(* LS Electric XG5000 project: QT(230517) *)
(* PLC NewPLC *)
(* module base 0 slot 0: FEnet:XGL-EFMT(B) (Fast Ethernet 통신 모듈, 전기 Master) *)
(* module base 1 slot 0: 아날로그입력 모듈:XGF-AC8A (A/D 전류 입력형 8채널) *)
(* module base 1 slot 1: 입력 모듈:XGI-D28A/B (DC 24V 입력, 64점 (전류소스 싱크공용/ 전류소스 입력)) *)
(* module base 1 slot 2: 입력 모듈:XGI-D28A/B (DC 24V 입력, 64점 (전류소스 싱크공용/ 전류소스 입력)) *)
(* module base 1 slot 3: 출력 모듈:XGQ-TR8A/B (트랜지스터 출력, 64점 (0.1A용, 싱크출력/소스출력)) *)
(* module base 1 slot 4: 출력 모듈:XGQ-TR8A/B (트랜지스터 출력, 64점 (0.1A용, 싱크출력/소스출력)) *)
(* module base 1 slot 5: Cnet:XGL-CH2A/B (Cnet 통신 모듈(RS-232C, RS-422/485)) *)
VAR_GLOBAL
    C485 : TON;
    C486 : TON;
    C487 : TON;
    TCPIP : TON;
    _0000_STAND_ALONE AT %LX60144 : BOOL; (* FEnet: 연결 안된 상태(Ver 6.0이상) *)
    _0100_CH0_ACT AT %UX1.0.16 : BOOL; (* 아날로그입력 모듈: 채널0 운전중 *)
    _0100_CH0_DATA AT %UW1.0.2 : INT; (* 아날로그입력 모듈: 채널0 변환값 *)
    _0100_CH0_IDD AT %UX1.0.160 : BOOL; (* 아날로그입력 모듈: 채널0 입력단선검출 *)
    _0100_CH1_ACT AT %UX1.0.17 : BOOL; (* 아날로그입력 모듈: 채널1 운전중 *)
    _0100_CH1_DATA AT %UW1.0.3 : INT; (* 아날로그입력 모듈: 채널1 변환값 *)
    _0100_CH1_IDD AT %UX1.0.161 : BOOL; (* 아날로그입력 모듈: 채널1 입력단선검출 *)
    _0100_CH2_ACT AT %UX1.0.18 : BOOL; (* 아날로그입력 모듈: 채널2 운전중 *)
    _0100_CH2_DATA AT %UW1.0.4 : INT; (* 아날로그입력 모듈: 채널2 변환값 *)
    _0100_CH2_IDD AT %UX1.0.162 : BOOL; (* 아날로그입력 모듈: 채널2 입력단선검출 *)
    _0100_CH3_ACT AT %UX1.0.19 : BOOL; (* 아날로그입력 모듈: 채널3 운전중 *)
    _0100_CH3_DATA AT %UW1.0.5 : INT; (* 아날로그입력 모듈: 채널3 변환값 *)
    _0100_CH3_IDD AT %UX1.0.163 : BOOL; (* 아날로그입력 모듈: 채널3 입력단선검출 *)
    _0100_CH4_ACT AT %UX1.0.20 : BOOL; (* 아날로그입력 모듈: 채널4 운전중 *)
    _0100_CH4_DATA AT %UW1.0.6 : INT; (* 아날로그입력 모듈: 채널4 변환값 *)
    _0100_CH4_IDD AT %UX1.0.164 : BOOL; (* 아날로그입력 모듈: 채널4 입력단선검출 *)
    _0100_CH5_ACT AT %UX1.0.21 : BOOL; (* 아날로그입력 모듈: 채널5 운전중 *)
    _0100_CH5_DATA AT %UW1.0.7 : INT; (* 아날로그입력 모듈: 채널5 변환값 *)
    _0100_CH5_IDD AT %UX1.0.165 : BOOL; (* 아날로그입력 모듈: 채널5 입력단선검출 *)
    _0100_CH6_ACT AT %UX1.0.22 : BOOL; (* 아날로그입력 모듈: 채널6 운전중 *)
    _0100_CH6_DATA AT %UW1.0.8 : INT; (* 아날로그입력 모듈: 채널6 변환값 *)
    _0100_CH6_IDD AT %UX1.0.166 : BOOL; (* 아날로그입력 모듈: 채널6 입력단선검출 *)
END_VAR

(* Comments on direct variables
%IX1.1.0	TK-301 HLV-PB
%IX1.1.1	P301ATR
%IX1.1.2	P301A Local sw
%IX1.1.3	P12AB
%IX1.1.4	LPB1AO
%IX1.1.5	P301A stop-PB
%IX1.1.6	P301A run-PB
%IX1.1.7	P301BTR
%IX1.1.8	P301B Local sw
%IX1.1.9	LPB1BF
%IX1.1.10	LPB1BO
%IX1.1.11	P301B stop-PB
%IX1.1.12	P301B Run PB
%IX1.1.13	P301CTR
%IX1.1.14	P301C Local sw
%IX1.1.15	LPB1CF
%IX1.1.16	LPB1CO
%IX1.1.17	P301C stop-PB
%IX1.1.18	P301C Run PB
%IX1.1.19	TK301-Clearance
%IX1.1.20	TK301-LEK
%IX1.1.21	P301ATH
%IX1.1.22	P301BTH
%IX1.1.23	P301CTH
%IX1.1.24	PUMP Room
%IX1.1.25	TK-302 HLV-PB
%IX1.1.26	  P302A  Trouble
%IX1.1.27	 P302A  LOCAL SW
%IX1.1.28	LPB2AF
%IX1.1.29	LPB2AO
%IX1.1.30	P302A stop-PB
%IX1.1.31	P302A run-PB
%IX1.1.32	  P302B  Trouble
%IX1.1.33	 P302B  LOCAL SW
%IX1.1.34	LPB2BF
%IX1.1.35	LPB2BO
%IX1.1.36	P302B stop-PB
%IX1.1.37	P302B run-PB
%IX1.1.38	  P302C  Trouble
%IX1.1.39	P302C  Local SW
%IX1.1.40	LPB2CF
%IX1.1.41	LPB2CO
%IX1.1.42	P302C stop-PB
%IX1.1.43	P302C run-PB
%IX1.1.44	TK302-Clearance
%IX1.1.45	TK302-LEK
%IX1.1.46	P302ATH
%IX1.1.47	P302BTH
%IX1.1.48	P302CTH
%IX1.1.49	TK-302 EM
%IX1.1.50	HLVD
(H30201)
%IX1.1.51	W30201
%IX1.1.52	  P303  Trouble
%IX1.1.53	P303  Local SW
%IX1.1.54	EMS1X
%IX1.1.55	EMS2X
%IX1.1.56	P303 stop-PB
%IX1.1.57	P303 Run PB
%IX1.1.58	Drain-303
Clearance
%IX1.1.59	EMS3X
%IX1.1.60	EMS4X
%IX1.1.61	P301A  1차 선택 SWITCH  (PANEL)
%IX1.1.62	P301B 1차 선택 SWITCH  (PANEL)
%IX1.1.63	P302A 1차 선택 SWITCH  (PANEL)
%IX1.2.0	P302B 1차 선택 SWITCH  (PANEL)
%IX1.2.1	P-301A 2차-PB
%IX1.2.2	P-301B 2차-PB
%IX1.2.3	P-302A 2차-PB
%IX1.2.4	P-302B 2차-PB
%IX1.2.5	Power-off PB
%IX1.2.6	Power-on PB
%IX1.2.7	Manual-PB
%IX1.2.8	Auto-PB
%IX1.2.9	AUTO START P/B
%IX1.2.10	Lamp-test PB
%IX1.2.11	AUTO STOP (PANEL)
%IX1.2.12	Horn Stop Panel
%IX1.2.13	EM_Reset
[Panel]
%IX1.2.14	PLC-Stanby operation
%IX1.2.16	운전선택 SCADA OR PANEL
%IX1.2.17	PANEL EM
%IX1.2.18	EMS1_C22
%IX1.2.19	EMS2_C21
%IX1.2.20	EMS3_C20
%IX1.2.21	EMS4_C19
%IX1.2.22	Cam1_R1
%IX1.2.23	Cam2_R2
%IX1.2.24	Cam3_R3
%IX1.2.25	BCVF
%IX1.2.26	TLV1
%IX1.2.27	TLV2
%IX1.2.28	TLV3
%IX1.2.29	TLV4
%IX1.2.32	SHELTURN1 TLV
%IX1.2.33	SHELTURN2 TLV
%IX1.2.34	SHELTURN3 TLV
%IX1.2.35	SHELTURN4 TLV
%IX1.2.36	P301A FS 
%IX1.2.37	P301B FS 
%IX1.2.38	P301C FS 
%IX1.2.39	P302A FS 
%IX1.2.40	P302B FS 
%IX1.2.41	P302C FS 
%IX1.2.42	P303 FS 
%IX1.2.43	P301A MC ON SIG 
%IX1.2.44	P301B MC ON SIG 
%IX1.2.45	P301C MC ON SIG 
%IX1.2.46	P302A MC ON SIG 
%IX1.2.47	P302B MC ON SIG 
%IX1.2.48	P302C MC ON SIG 
%IX1.2.49	P303 MC ON SIG 
%IX1.2.56	HLVB(하차 VALVE)
%IX1.3.0	PL29-R
%IX1.3.1	L37-Y
%IX1.3.48	TK-110 HLV 선택PB
%IX2.3.1	P101A THERMOSTAT
%ID1.0.0	디지털_입력
%QX1.3.0	TK-301 HLV on
%QX1.3.1	P301A Trouble
%QX1.3.2	  P301A  Local
%QX1.3.3	P301A-stop Lamp
%QX1.3.4	P301A Run
%QX1.3.5	P301B-Trouble
%QX1.3.6	P301B- Local
%QX1.3.7	P301B-stop
%QX1.3.8	P301B Run
%QX1.3.9	P301C-Trouble
%QX1.3.10	P301C- Local
%QX1.3.11	P301C-stop Lamp
%QX1.3.12	P301C Run
%QX1.3.13	TK-301 HH
%QX1.3.14	TK-301 H
%QX1.3.15	TK-301 ATG TROUBLE
%QX1.3.16	TK-301 L
%QX1.3.17	TK-301 LL
%QX1.3.18	TK-301 Leakage
%QX1.3.19	TK-302 HLV on
%QX1.3.20	P302A Trouble
%QX1.3.21	  P302A   Local
%QX1.3.22	P302A  Stop Lamp
%QX1.3.23	P302A Run
%QX1.3.24	P302B-Trouble
%QX1.3.25	  P302B   Local
%QX1.3.26	P302B  Stop Lamp
%QX1.3.27	P302B Run
%QX1.3.28	P302C-Trouble
%QX1.3.29	  P302C  Local
%QX1.3.30	P302C  Stop Lamp
%QX1.3.31	P302C Run
%QX1.3.32	TK-302 HH
%QX1.3.33	TK-302 H
%QX1.3.34	TK-302 ATG TROUBLE
%QX1.3.35	TK-302 L
%QX1.3.36	TK-302 LL
%QX1.3.37	TK-302 Leakage
%QX1.3.38	TK-303 HLVD
%QX1.3.39	TK-303 Water
%QX1.3.40	P303-Trouble lamp
%QX1.3.41	  P303  Local
%QX1.3.42	P303  Stop Lamp
%QX1.3.43	P303 Run
%QX1.3.44	TK-303 Max2
%QX1.3.45	TK-303_LT33_H
%QX1.3.46	TK-303 Nomal
%QX1.3.47	TK-303 Min1
%QX1.3.48	TK-303 Min2
%QX1.3.49	P301A 1차 선택 Lamp
%QX1.3.50	P301A 2차 선택 Lamp
%QX1.3.51	P301B 1차 선택 Lamp
%QX1.3.52	P301B 2차 선택 Lamp
%QX1.3.53	P302A 1차 선택 Lamp
%QX1.3.54	P302A 2차 선택 Lamp
%QX1.3.55	P302B 1차 선택 Lamp
%QX1.3.56	P302B 2차 선택 Lamp
%QX1.3.57	Power-off LAMP
%QX1.3.58	Power-on LAMP
%QX1.3.59	Manual LAMP
%QX1.3.60	Auto 선택 LAMP
%QX1.3.61	AUTO START LAMP
%QX1.3.62	AUTO STOP LAMP
%QX1.3.63	압력저하 (PT-301)
%QX1.4.0	Horn Stop Lamp
%QX1.4.1	Pump-start 6time/h
%QX1.4.2	BPCV1-Lamp
%QX1.4.3	CVP-Lamp
%QX1.4.4	EV-Lamp
%QX1.4.5	EM RESET LAMP
%QX1.4.6	BCVF-Lamp
%QX1.4.7	Lamp_test LAMP
%QX1.4.8	PUMP Room
%QX1.4.9	EM-Panel
%QX1.4.10	Shelter-1
%QX1.4.11	Shelter-2
%QX1.4.12	Shelter-3
%QX1.4.13	Shelter-4
%QX1.4.14	Emergency-local
%QX1.4.15	PIT1-Trouble 
%QX1.4.16	PIT2-Trouble 
%QX1.4.17	FIT1-Trouble 
%QX1.4.18	FIT2-Trouble 
%QX1.4.19	FIT3-Trouble 
%QX1.4.20	FIT4-Trouble 
%QX1.4.21	MASTER PLC LAMP
%QX1.4.22	Control-unit 1 Trouble
%QX1.4.23	STANDBY PLC LAMP
%QX1.4.24	Control-unit 2 Trouble
%QX1.4.25	Horn Relay
%QX1.4.26	PUMP Room
%QX1.4.27	TK-302 EM
%QX1.4.28	Panel 선택 Lamp
%QX1.4.29	SCADA 선택 Lamp
%QX1.4.30	BPCV1-Sol
%QX1.4.31	BPCV2-Sol
%QX1.4.32	CVP SOL
%QX1.4.33	EV-Sol
%QX1.4.34	R1_PT3-4/PT5-6
%QX1.4.35	R2_FT1-2/FT5-6
%QX1.4.36	R2_FT3-4/FTT-8
%QX1.4.37	TK-301 HLV OPEN LAMP
%QX1.4.38	P301A Run LAMP
%QX1.4.39	P301B Run LAMP
%QX1.4.40	P301C Run LAMP
%QX1.4.41	TK-302 HLV OPEN LAMP
%QX1.4.42	P302A Run LAMP
%QX1.4.43	P302B Run LAMP
%QX1.4.44	P302C Run LAMP
%QX1.4.45	P303 Run LAMP
%QX1.6.2	SCADA 선택 Lamp
%QX1.6.3	Panel 선택 Lamp
%QX2.2.26	출하 PUMP P101A 1차 운전 선택 Lamp
%QX2.2.27	출하 PUMP P101B 1차 운전 선택 Lamp
%QX2.2.42	출하 PUMP P101A 2차 운전 선택 Lamp
%QX2.2.43	출하 PUMP P101B 2차 운전 선택 Lamp
%MX0	P301A_Run
%MX1	P301B_Run
%MX2	P301A_Pump
%MX3	P301A_FS
%MX5	P301A_Trouble
%MX6	TK-301 HLV,P301A,P301B_Run
%MX7	P301A,OR P301B_RUN
%MX8	P301B_Pump
%MX9	P301B_FS
%MX10	P301A_P301B_ Trouble
%MX12	BPCV_On
%MX14	P301B_Trouble
%MX15	P301C_RUN
%MX16	P301C_STOP
%MX17	P301C_PUMP
%MX18	QT_BOTTOM TAP COLOR(X PUMP RUN)
%MX19	TK-302 HLV,P302A,P302B_Run
%MX20	P302A_Run
%MX21	P302A,OR P302B_RUN
%MX22	P302A_Pump
%MX23	P302A_FS
%MX24	P302A_Trouble
%MX25	P302B_Run
%MX26	P302A_P302B_ Trouble
%MX27	P302B-Pump
%MX28	P302B_FS
%MX29	P302B_Trouble
%MX30	P302C_Run
%MX31	P301 회수중
%MX32	P302C_Pump
%MX33	P302C_FS
%MX34	P302C_Trouble
%MX35	P303_Run
%MX36	P302 회수중
%MX37	P303_Pump
%MX38	P303_FS
%MX39	P303_Trouble
%MX40	Alarm Reset
%MX45	TLV1
%MX46	TLV2
%MX47	TLV3
%MX48	TLV4
%MX49	HLV1
%MX50	HLV2
%MX51	TK-301 출하
%MX52	출하_EV
%MX53	출하_CVP
%MX54	출하_BPCV
%MX55	회수라인
%MX56	TK301_회수
%MX57	TK302_회수
%MX58	QT01_출하
%MX59	QT02_출하
%MX60	QT03_출하
%MX61	QT04_출하
%MX62	AUTO START OK
%MX65	TLV1
%MX66	TLV2
%MX67	TLV3
%MX68	TLV4
%MX79	TK-104 선택 SCADA    (수령)
%MX82	QT_TANK_HH
%MX100	TK-301 CH0 단선
%MX101	TK-301 Min2
%MX102	TK-301 Min1
%MX103	TK-301 Max1
%MX104	TK-301 Max2
%MX105	TK-302 CH1 단선
%MX106	TK-302 Min2
%MX107	TK-302 Min1
%MX108	TK-302 Max1
%MX109	TK-302 Max2
%MX110	TK-303 CH1 단선
%MX111	TK-303 Min2
%MX112	TK-303 Min1
%MX113	TK-303 Max1
%MX114	TK-303 Max2
%MX128	P301A run-PB  (SCADA)
%MX129	P301A stop-PB  (SCADA)
%MX130	Manual_Scada
%MX131	Auto_Scada
%MX132	P301B Run PB(SCADA)
%MX133	P301B stop-PB(SCADA)
%MX134	  AUTO   START  (SCADA)
%MX135	AUTO STOP (SCADA)
%MX136	P301C Run PB(SCADA)
%MX137	P301C stop-PB(SCADA)
%MX138	P302A Run PB(SCADA)
%MX139	P302A stop-PB(SCADA)
%MX140	P302B Run PB(SCADA)
%MX141	P302B stop-PB(SCADA)
%MX142	P302C Run PB(SCADA)
%MX143	P302C stop-PB(SCADA)
%MX144	P303 Run PB(SCADA)
%MX145	P303 stop-PB(SCADA)
%MX146	EM-Reset
[SCADA]
%MX147	Horn Stop SCADA
%MX148	P301A Lock key Run
%MX149	P301B Lock key Run
%MX150	P301C Lock key Run
%MX151	P302A Lock key Run
%MX152	P302B Lock key Run
%MX153	P302C Lock key Run
%MX154	P303 Lock key Run
%MX160	이글루#1유량 - 값
%MX161	이글루#2유량 - 값
%MX162	이글루#3유량 - 값
%MX163	이글루#4유량 - 값
%MX164	수령 유량 -값
%MX169	L5 BPCV
%MX170	L6 CVP
%MX171	L7 BCVF (By-Pass Valve)
%MX172	L8 EV
%MX173	수령유량 - 값
%MX177	TK-303_LT33_FAULT
%MX180	P303_Remote
%MX181	P303_Stop
%MX182	P303_Run
%MX183	P303_Fault
%MX184	P303_F.S
%MX185	P303_O.L
%MX186	P303_HLVD
%MX192	TK-301 HLV SCADA ON
%MX193	TK-302 HLV SCADA ON
%MX206	TK-301 ATG NO SIGNAL
%MX207	TK-301_LL
%MX208	TK-301_LT31_L
%MX209	TK-301_LT31_H
%MX210	TK-301_HH_SIG
%MX212	P301A_Key
%MX213	P301A_Remote
%MX214	P301A_Stop
%MX215	P301A_Run
%MX216	P301A_Fault
%MX217	P301A FS_Fault
%MX218	P301A_O.L
%MX219	P301B_Key
%MX220	301B_Remote
%MX221	P301B_Stop
%MX222	P301B_Run
%MX223	P301B_Fault
%MX224	P301B_F.S
%MX225	P301B_O.L
%MX226	P301C_Remote
%MX227	P301C_Stop
%MX228	P301C_Run
%MX229	P301C_Fault
%MX235	TK-302_LL
SIG
%MX236	TK-302 L
SIG
%MX237	TK-302_H
_SIG
%MX238	TK-302_HH_SIG
%MX239	TK-302 ATG NO SIGNAL
%MX240	P302A_Key
%MX241	P302A_Remote
%MX242	P302A_Stop
%MX243	P302A_Run
%MX244	P302A_Fault
%MX245	P302A_F.S
%MX246	P302A_O.L
%MX247	P302B_Key
%MX248	P302B_Remote
%MX249	P302B_Stop
%MX250	P302B_Run
%MX251	P302B_Fault
%MX252	P302B_F.S
%MX253	P302B_O.L
%MX254	P302C_Remote
%MX255	P302C_Stop
%MX256	P302C_Run
%MX257	P302C_Fault
%MX263	PRI1_301A
%MX264	PRI1_301B
%MX265	PRI1_302A
%MX266	PRI1_302B
%MX267	PRI2_301A
%MX268	PRI2_301B
%MX269	PRI2_302A
%MX270	PRI2_302B
%MX272	CH1 PIT3-4 Trouble
%MX273	CH2 FT301 Trouble
%MX274	CH3 FIT3-4 Trouble
%MX277	CH3 FT-302 Trouble
%MX301	P-301A 1차-out
%MX303	P-301B 1차-out
%MX305	P-302A 1차-out
%MX307	P-302B 1차-out
%MX309	P-301A 2차-out
%MX310	P-301B 2차-on
%MX312	P-302A 2차-on
%MX313	TANK101 LEVEL 15%   L
%MX314	P-302B 2차-on
%MX330	TK-303_HH
%MX331	TK-303_H
%MX332	TK-303_ATG TROUBLE
%MX333	TK-303_L
%MX334	TK-303_LL
%MX335	QT_NMR#3
SIGNAL OFF 
ALARM
%MX340	P301A 1차 선택
%MX341	P301B 1차 선택
%MX342	P302A 1차 선택
%MX343	P302B 1차 선택
%MX344	P301A 2차 선택
%MX345	P301B 2차 선택
%MX346	P302A 2차 선택
%MX347	P302B 2차 선택
%MX352	P012A 2차 선택
%MX353	P012B 2차 선택
%MX360	P012A 1차 선택
%MX361	P021B 1차 선택
%MX362	P021A 2차 선택
%MX363	P021B 2차 선택
%MX398	1차 펌프 작동
%MX399	1차 펌프정지 압력
%MX400	Auto Run SIG
%MX401	1차 펌프 정지
%MX402	1차 펌프 초기 기동 압력
%MX403	1차 회수유량
%MX404	2차 펌프 작동
%MX405	1차 회수유량
%MX406	2차 회수유량
%MX407	2차 펌프정지
%MX408	1차 정지유량
%MX409	1차 재기동방지
%MX412	2차 펌프 정지
%MX413	1차 펌프정지 SIG
%MX414	1차 펌프 정지
%MX448	P301A  1차 선택 SWITCH  (SCADA)
%MX449	P301B 1차 선택 SWITCH  (SCADA)
%MX450	P301A 2차 선택 SWITCH  (SCADA)
%MX451	P301B 2차 선택 SWITCH  (SCADA)
%MX452	P302A 1차 선택 SWITCH  (SCADA)
%MX453	P302B 1차 선택 SWITCH  (SCADA)
%MX454	P302A 2차 선택 SWITCH  (SCADA)
%MX455	P302B 2차 선택 SWITCH  (SCADA)
%MX456	선택완료  (SCADA)
%MX458	P012A  1차 선택 SWITCH  (SCADA)
%MX459	P012B  1차 선택 SWITCH  (SCADA)
%MX460	P012A  2차 선택 SWITCH  (SCADA)
%MX461	P012B  2차 선택 SWITCH  (SCADA)
%MX468	P021A  1차 선택 SWITCH  (SCADA)
%MX469	P021B 1차 선택 SWITCH  (SCADA)
%MX470	P021A  2차 선택 SWITCH  (SCADA)
%MX471	P021B 2차 선택 SWITCH  (SCADA)
%MX500	통신 쓰기 PULS
%MX501	통신 읽기 PULS
%MX511	Auto_ P-301A_ON_REQ
%MX512	Scada_auto
%MX513	Scada_man
%MX514	S-P301A manual Run
%MX515	S-P301B manual Run
%MX516	S-P301C manual Run
%MX517	S-P302A manual Run
%MX518	S-P302B manual Run
%MX519	S-P302C manual Run
%MX520	S-P303 manual Run
%MX528	Shelturn4-Em
%MX529	Total Emergency
%MX530	 Total Alarm
%MX531	Horn Stop
%MX532	TK-301 HLV on-off
%MX533	TK-302 HLV on-off
%MX534	CVP_on
%MX536	HLV21201 TK110 OPEN PULS(MANU)
%MX537	Any HLV Open
%MX538	TK-302 Interlock 
%MX539	TK-301 Interlock 
%MX543	P-301A 1차_off
%MX544	P-301A 1차_out
%MX545	P-301B 1차_off
%MX546	P-301B 1차_out
%MX547	P-302A 1차_off
%MX548	P-302A 1차_out
%MX549	P-302B 1차_off
%MX550	P-302B 1차_out
%MX551	P-301A 2차_off
%MX552	P-301A 2차_out
%MX553	P-301B 2차_off
%MX554	P-301B 2차_out
%MX555	P-302A 2차_off
%MX556	P-302A 2차_out
%MX557	P-302B 2차_off
%MX558	P-302B 2차_out
%MX561	TK301 Auto
1차 
펌프운전중 
%MX562	Auto-1차 펌프정지 
%MX563	TK301 Auto
2차 
펌프운전중 
%MX564	Auto-2차 펌프정지 
%MX565	Auto P-301A_ON
%MX566	Auto P-301B_ON
%MX567	Auto P-302A_ON
%MX568	Auto P-302B_ON
%MX581	TK302 Auto
1차 
펌프운전중 
%MX591	TK302 Auto
2차 
펌프운전중 
%MX592	Auto_2차 펌프정지
%MX593	자동운전 시작
%MX594	펌프정지 압력
%MX595	Auto Run
%MX596	자동운전 정지
%MX597	1-2차 펌프on
%MX598	2차 펌프준비
%MX599	2차 펌프on
%MX600	1차 회수유량
%MX601	2차 회수유량
%MX602	2차 펌프정지
%MX603	1차 정지유량
%MX604	1차 재기동방지
%MX605	2차 펌프정지
%MX606	1차 펌프정지
%MX607	펌프운전 Rest
%MX640	PUMP Room
%MX641	TK-302 Em 사용안함
%MX642	TK-301 & 302 Em
%MX643	Panel-Em
%MX644	Shelturn1-Em
%MX645	Shelturn2-Em
%MX646	Shelturn3-Em
%MX647	Shelturn4-C19
%MX648	Local EM
%MX649	EMS1X
%MX650	EMS2X
%MX651	EMS3X
%MX652	EMS4X
%MX656	RS-485 통신이상
%MX657	TCPIP 통신이상
%MX1010	모드버스 브럭1-1 동작
%MX1200	모드버스 브럭2-1 동작
%MX1220	모드버스 브럭2-2 동작
%MX1300	모드버스 브럭3-1 동작
%MX1320	모드버스 브럭3-2 동작
%MX1400	모드버스 브럭4-1 동작
%MX1420	모드버스 브럭4-2 동작
%MX1500	모드버스 브럭5-1 동작
%MX1520	모드버스 브럭5-2 동작
%MX3232	이중화운전_A_Side_MASTER
%MX3233	이중화운전_B_Side_MASTER
%MX3234	A-Side 단독운전
%MX3235	B-Side 단독운전
%MX4816	AUTO HLV_301 OPEN
%MX4832	AUTO HLV_302 OPEN
%MX6400	Panel Manual
%MX6401	SCADA Manual
%MX6402	Panel Auto
%MX6403	SCADA Auto
%MX6405	BUZZER STOP
%MX6410	Manual 선택
%MX6411	Auto 선택
%MX6464	LAMP TEST SIG
%MX6476	MAIN PNL-EM
%MX10002	TEST2
%MX12800	AUTO START OK
%MX12801	AUTO STOP OK
%MX19200	P301A ALARM
%MX19201	P301A FS ALARM
%MX19202	P301B ALARM
%MX19203	P301B FS ALARM
%MX19204	P301C ALARM
%MX19205	P301C FS ALARM
%MX19206	P302A ALARM
%MX19207	P302A FS ALARM
%MX19208	P302B ALARM
%MX19209	P302B FS ALARM
%MX19210	P302C ALARM
%MX19211	P302C FS ALARM
%MX19212	P303 
ALARM
%MX19213	P303 FS ALARM
%MX19215	P301A FS SIG
%MX19216	P301B FS SIG
%MX19217	P301C FS SIG
%MX19218	P302A FS SIG
%MX19219	P302B FS SIG
%MX19220	P302C FS SIG
%MX19221	P303 FS SIG
%MX19264	P301A 수동 RUN
%MX19265	P301B 수동 RUN
%MX19266	P301C 수동 RUN
%MX19267	P302A 수동 RUN
%MX19268	P302B 수동 RUN
%MX19269	P302C 수동 RUN
%MX19270	P303 수동 RUN
%MX19905	P301A 1차 작동
%MX19906	P301A 2차 작동
%MX19969	P301B 1차 작동
%MX19970	P301B 2차 작동
%MX20545	P302A 1차 작동
%MX20546	P302A 2차 작동
%MX20609	P302B 1차 작동
%MX20610	P302B 2차 작동
%MX23087	Auto start all ready
%MX23089	ARES Stop SIG
%MX23680	TK-301 수령 송유관 색변화
%MX23681	TK-301  불출 송유관 색변화
%MX23682	TK-301,302 수령 송유관 색변화 
%MX23683	TK-301,302 불출 송유관 색변화
%MX23684	TK-302 수령 송유관 색변화
%MX23685	TK-302 불출 송유관 색변화 2
%MX23686	TK-301C,302C DRAIN 송유관 색변화
%MX23687	TK-302 DRAIN 송유관 색변화
%MX23688	SHELTURN1 송유관 색변화1 
%MX23689	SHELTURN2 송유관 색변화 2
%MX23690	SHELTURN3 송유관 색변화
%MX23691	SHELTURN4 송유관 색변화
%MX25600	AUTO START OK
%MX25602	ALL REMOTE
%MX25665	P101A Auto 2차 Run
%MX25666	P101B Auto 1차 Run
%MX25667	P101B Auto 2차 Run
%MX26112	QT_Auto_2st_Pump Run
%MX26113	QT_Auto_restart_alarm[TLV_SIG]
%MX26240	1차 PUMP Running Timing
%MX26241	2차 PUMP Running Timing
%MX26242	1차 PUMP Stoping
%MX26243	2차 PUMP Stoping
%MX26244	Auto Run BPCV Stop
%MX26246	1차 펌프 정지조건 홀딩
%MX26247	헌팅 보정
%MX26250	1차 PUMP Stoping 조건
%MX26256	holding pressure charge
%WW0	C22_BCU STATUS
%WW1	C22 BCU STATUS VALUE
%WW2	C21_BCU STATUS
%WW3	C20 BCU STATUS VALUE
%WW4	C20 BCU STATUS
%WW5	C20 BCU STATUS VALUE
%WW6	C19 BCU STATUS
%WW7	C19 BCU STATUS VALUE
%WW10	 P301 1차 선택 SET
%WW11	1차 선택 SET
%WW12	2차 선택 SET
%WW13	 P302 2차 선택 SET
%WW20	TANK301 문자열
%WW21	TK-302 문자열
%WW102	TK-301 LEVEL (PLC -> SCADA)
%WW150	P301A RUN SET
%WW151	P301B RUN SET
%WW152	P301C RUN SET
%WW153	P302A RUN SET
%WW154	P302B RUN SET
%WW155	P302C RUN SET
%WW156	P303 RUN SET
%WW202	TK-302 LEVEL (PLC -> SCADA)
%WW211	TK-112 H SET
%WW310	TK-301 HH SET
%WW311	TK-301 H SET
%WW312	TK-301 L SET
%WW313	TK-301 LL SET
%WW320	TK-302 HH SET
%WW321	TK-302 H SET
%WW322	TK-302 L SET
%WW323	TK-302 LL SET
%WW330	TK-303 HH SET
%WW331	TK-303 H SET
%WW332	TK-303 L SET
%WW333	TK-303 LL SET
%WW440	불출유량 - 회수유량 = 값
%WW500	TK301Level NRM500 - >PLC
%WW501	Error Status Ref.TK301
[NMR#3]
word
%WW503	TK302Level(NRM5000 ->PLC)
%WW504	Error Status Ref.TK302
[NMR#3]
word
%WW506	DRAIN TANK TK-111 LEVEL (PLC -> SCADA)
%WW682	TK-301 VOLUME (CTM->PLC)
%WW690	TK303 VOLUME(커텀스->PLC)
%WW691	TK111 VOLUME(커텀스->PLC)
%WW1000	이글루 #1 유량(High)
%WW1001	이글루 #1 유량(Low)
%WW1020	이글루 #2 유량(High)
%WW1021	이글루 #2 유량(Low)
%WW1040	이글루 #3 유량(High)
%WW1041	이글루 #3 유량 (Low)
%WW1060	이글루 #4 유량(high)
%WW1061	이글루 #4 유량(Low)
%WW1080	수령 유량
(High)
%WW1081	수령 유량 (Low)
%WW1100	PT301 출하압력 값
%WW1102	PT301출하압력 PSI
%WW1200	FT301 출하유량 값
%WW1202	FT301출하유량 GPM
%WW1204	FT301 출하유량
%WW1300	FT302 회수유량 값
%WW1302	FT302회수유량 GPM
%WW1304	FT302 회수유량
%WW1400	TK_303 변환값
%WW1402	TK-303 LEVEL (PLC -> SCADA)
%WW1404	DRAIN TANK TK-303 LEVEL (PLC -> CTM)
%WW1502	QT TLV 
COUNT
%WW1600	QT_TLV_EA
%WW1601	AUTO 
TK-301 HLV OPEN SIG
%WW1602	TK-302 HLV
OPEN SIG
%WW2000	이글루#1 BCU Command
%WW2002	이글루#2 BCU Command
%WW2004	이글루#3 BCU Command
%WW2006	이글루#4 BCU Command
%WD532	Total of Gross_AUX
%WD534	Total of Net_AUX
%WD536	Total of Mass_AUX
%WD538	Total of Acc, Gross_AUX
%WD540	Rate of Gross_AUX
%WD542	Batch Preset [0]_AUX
%WD544	Total of Gross_AUX
%WD546	Total of Net_AUX
%WD548	Total of Mass_AUX
%WD550	Total of Acc, Gross_AUX
%WD552	Rate of Gross_AUX
%WD554	Batch Preset [0]_AUX
%WD556	Total of Gross_AUX
%WD558	Total of Net_AUX
%WD560	Total of Mass_AUX
%WD562	Total of Acc, Gross_AUX
%WD564	Rate of Gross_AUX
%WD566	Batch Preset [0]_AUX
%WD568	Total of Gross_AUX
%WD570	Total of Net_AUX
%WD572	Total of Mass_AUX
%WD574	Total of Acc, Gross_AUX
%WD576	Rate of Gross_AUX
%WD578	Batch Preset [0]_AUX
%WD600	Total of Gross
%WD602	Total of Net
%WD604	Total of Mass
%WD606	Total of Acc, Gross
%WD608	Rate of Gross
%WD610	Batch Preset [0]
%WD650	Total of Gross
%WD652	Total of Net
%WD654	Total of Mass
%WD656	Total of Acc, Gross
%WD658	Rate of Gross
%WD660	Batch Preset [0]
%WD686	TK-302 VOLUME (SCADA => PLC)
%WD690	TK-303 VOLUME (SCADA => HS)
%WD700	Total of Gross
%WD702	Total of Net
%WD704	Total of Mass
%WD706	Total of Acc, Gross
%WD708	Rate of Gross
%WD710	Batch Preset [0]
%WD750	Total of Gross
%WD752	Total of Net
%WD754	Total of Mass
%WD756	Total of Acc, Gross
%WD758	Rate of Gross
%WD760	Batch Preset [0]
%WD1010	이글루 #1 Dword
%WD1012	이글루 #1 Float
%WD1013	이글루 #1 유량 값
%WD1020	이글루 #2 Dword
%WD1022	이글루 #2 Float
%WD1023	이글루 #2 유량 값
%WD1030	이글루 #3 Dword
%WD1032	이글루 #3 Float
%WD1033	이글루 #3 유량 값
%WD1040	이글루 #4 Dword
%WD1042	이글루 #4 Float
%WD1043	이글루 #4 유량 값
%WD1050	수령유량  Dword
%WD1052	수령유량 Float
%WD1053	수령유량  값
%WD1406	TK303_VOL (PLC -> SCADA)
%WD5100	Total of Gross
%WD5102	Total of Net
%WD5104	Total of Mass
%WD5106	Total of Acc.Gross
%WD5108	Rate of Gross
%WD5110	Batch of Press[0]
*)

PROGRAM Main (* task: 스캔 프로그램 *)
VAR
    CVP : TON;
    INST : TOF;
    L_TST : TON;
    L_TST_FS : TON;
    T8 : TON; (* CVP-delay10s *)
    T9 : TON; (* CVP-delay10s *)
END_VAR
VAR
    _p1 : BOOL;
    _p2 : BOOL;
END_VAR

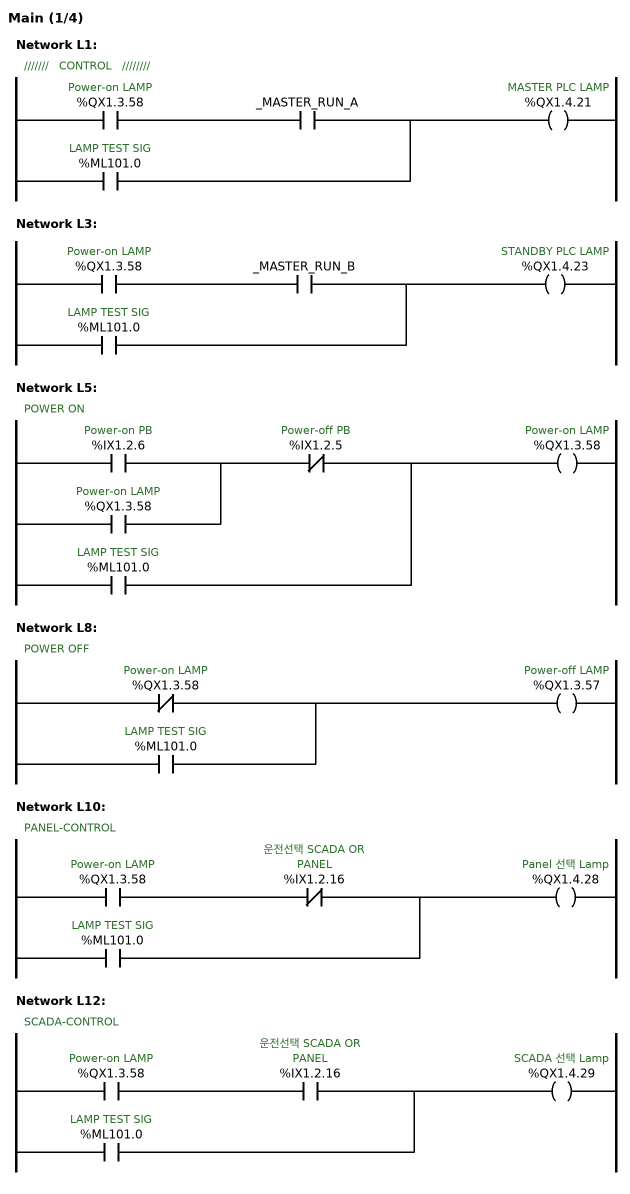
(* ///////   CONTROL   //////// *)
(* Rung L1 *)
%QX1.4.21 := (%QX1.3.58 AND _MASTER_RUN_A) OR %ML101.0;
(* Rung L3 *)
%QX1.4.23 := (%QX1.3.58 AND _MASTER_RUN_B) OR %ML101.0;
(* Rung L5 *)
%QX1.3.58 := ((%IX1.2.6 OR %QX1.3.58) AND NOT %IX1.2.5) OR %ML101.0;
(* POWER ON *)
(* Rung L8 *)
%QX1.3.57 := NOT %QX1.3.58 OR %ML101.0;
(* POWER OFF *)
(* Rung L10 *)
%QX1.4.28 := (%QX1.3.58 AND NOT %IX1.2.16) OR %ML101.0;
(* PANEL-CONTROL *)
(* Rung L12 *)
%QX1.4.29 := (%QX1.3.58 AND %IX1.2.16) OR %ML101.0;
(* SCADA-CONTROL *)

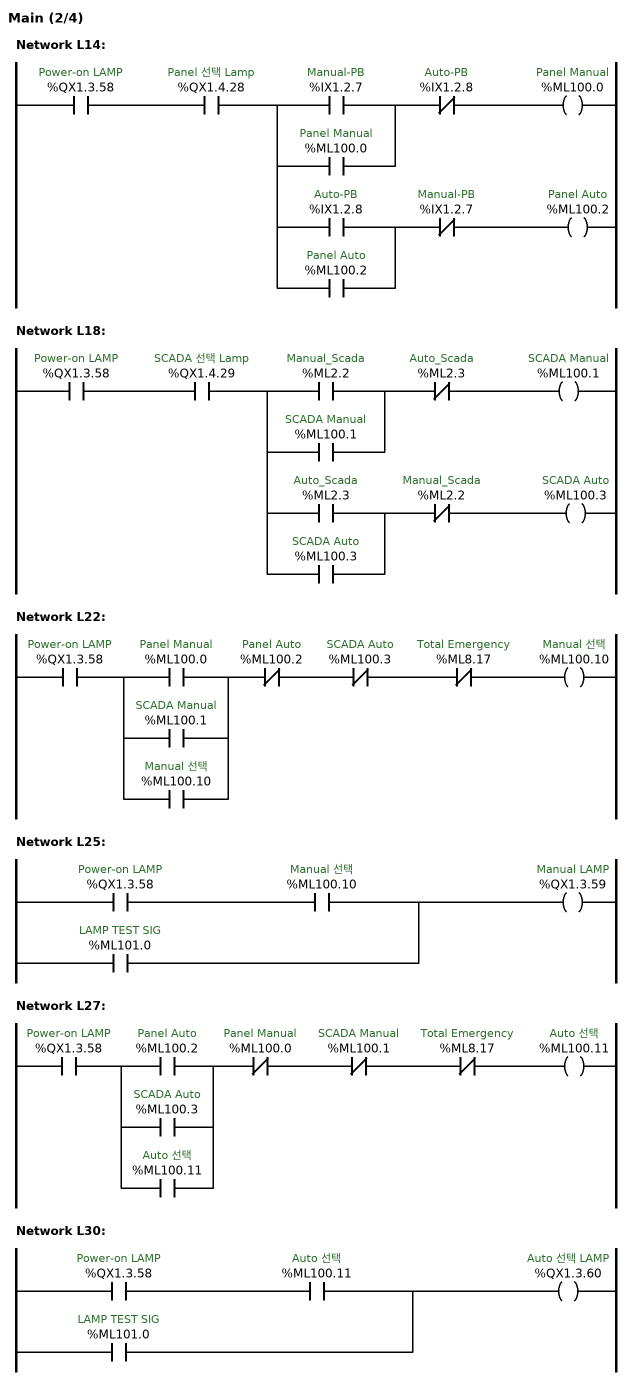
(* Rung L14 *)
%ML100.0 := %QX1.3.58 AND %QX1.4.28 AND (%IX1.2.7 OR %ML100.0) AND NOT %IX1.2.8;
%ML100.2 := %QX1.3.58 AND %QX1.4.28 AND (%IX1.2.8 OR %ML100.2) AND NOT %IX1.2.7;
(* Rung L18 *)
%ML100.1 := %QX1.3.58 AND %QX1.4.29 AND (%ML2.2 OR %ML100.1) AND NOT %ML2.3;
%ML100.3 := %QX1.3.58 AND %QX1.4.29 AND (%ML2.3 OR %ML100.3) AND NOT %ML2.2;
(* Rung L22 *)
%ML100.10 := %QX1.3.58 AND (%ML100.0 OR %ML100.1 OR %ML100.10) AND NOT %ML100.2 AND NOT %ML100.3 AND NOT %ML8.17;
(* Rung L25 *)
%QX1.3.59 := (%QX1.3.58 AND %ML100.10) OR %ML101.0;
(* Rung L27 *)
%ML100.11 := %QX1.3.58 AND (%ML100.2 OR %ML100.3 OR %ML100.11) AND NOT %ML100.0 AND NOT %ML100.1 AND NOT %ML8.17;
(* Rung L30 *)
%QX1.3.60 := (%QX1.3.58 AND %ML100.11) OR %ML101.0;

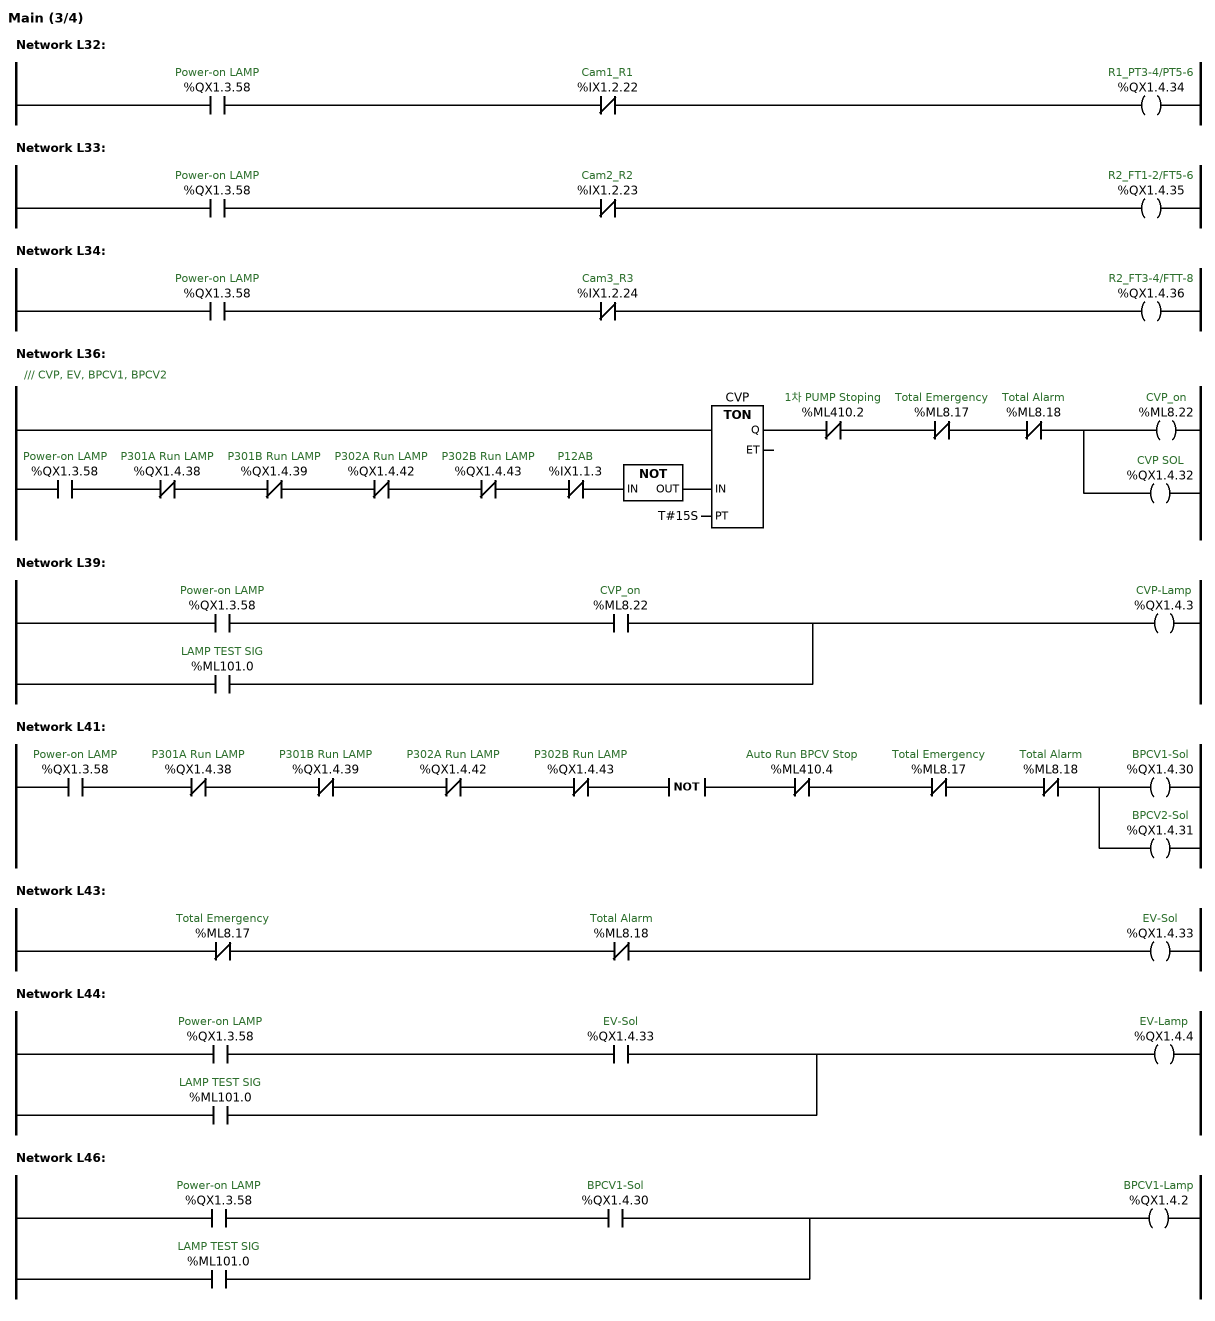
(* Rung L32 *)
%QX1.4.34 := %QX1.3.58 AND NOT %IX1.2.22;
(* Rung L33 *)
%QX1.4.35 := %QX1.3.58 AND NOT %IX1.2.23;
(* Rung L34 *)
%QX1.4.36 := %QX1.3.58 AND NOT %IX1.2.24;
(* /// CVP, EV, BPCV1, BPCV2 *)
(* Rung L36 *)
CVP(IN := NOT (%QX1.3.58 AND NOT %QX1.4.38 AND NOT %QX1.4.39 AND NOT %QX1.4.42 AND NOT %QX1.4.43 AND NOT %IX1.1.3), PT := T#15S);
_p1 := CVP.Q AND NOT %ML410.2 AND NOT %ML8.17 AND NOT %ML8.18;
%ML8.22 := _p1;
%QX1.4.32 := _p1;
(* Rung L39 *)
%QX1.4.3 := (%QX1.3.58 AND %ML8.22) OR %ML101.0;
(* Rung L41 *)
_p2 := NOT (%QX1.3.58 AND NOT %QX1.4.38 AND NOT %QX1.4.39 AND NOT %QX1.4.42 AND NOT %QX1.4.43) AND NOT %ML410.4 AND NOT %ML8.17 AND NOT %ML8.18;
%QX1.4.30 := _p2;
%QX1.4.31 := _p2;
(* Rung L43 *)
%QX1.4.33 := NOT %ML8.17 AND NOT %ML8.18;
(* Rung L44 *)
%QX1.4.4 := (%QX1.3.58 AND %QX1.4.33) OR %ML101.0;
(* Rung L46 *)
%QX1.4.2 := (%QX1.3.58 AND %QX1.4.30) OR %ML101.0;

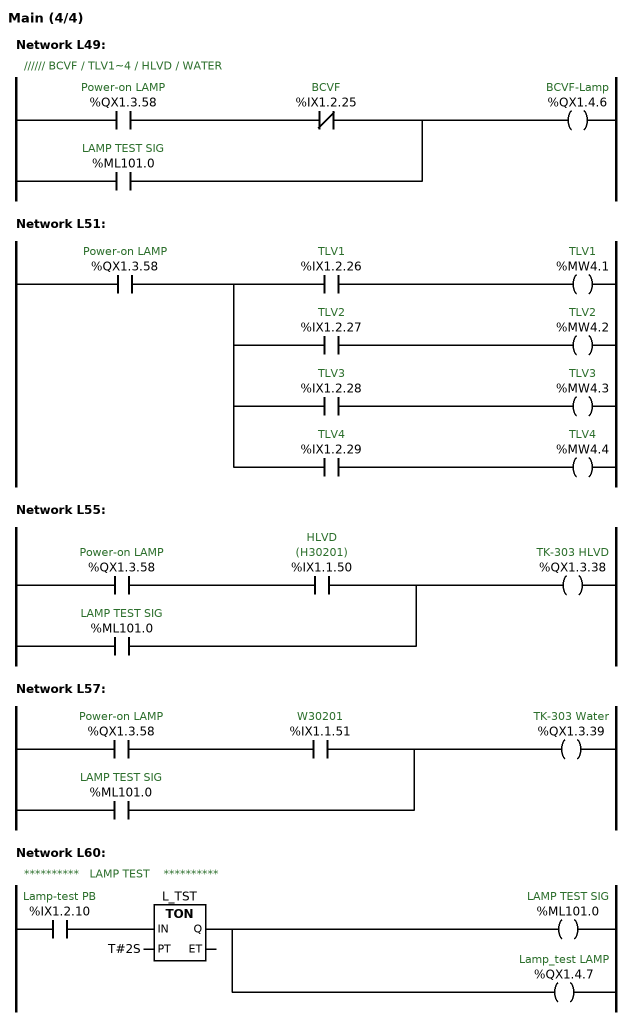
(* ////// BCVF / TLV1~4 / HLVD / WATER *)
(* Rung L49 *)
%QX1.4.6 := (%QX1.3.58 AND NOT %IX1.2.25) OR %ML101.0;
(* Rung L51 *)
%MW4.1 := %QX1.3.58 AND %IX1.2.26;
%MW4.2 := %QX1.3.58 AND %IX1.2.27;
%MW4.3 := %QX1.3.58 AND %IX1.2.28;
%MW4.4 := %QX1.3.58 AND %IX1.2.29;
(* Rung L55 *)
%QX1.3.38 := (%QX1.3.58 AND %IX1.1.50) OR %ML101.0;
(* Rung L57 *)
%QX1.3.39 := (%QX1.3.58 AND %IX1.1.51) OR %ML101.0;
(* **********   LAMP TEST    ********** *)
(* Rung L60 *)
L_TST(IN := %IX1.2.10, PT := T#2S);
%ML101.0 := L_TST.Q;
%QX1.4.7 := L_TST.Q;
END_PROGRAM

PROGRAM Manual (* task: 스캔 프로그램 *)
VAR
    Down_1 : CTD_INT; (* Down_1 *)
    INST : TON; (* INST *)
    INST1 : TON; (* INST1 *)
    INST2 : TON;
    INST3 : TON; (* INST1 *)
    OFF_Delay : TOF; (* Off_Delay *)
    ON_Delay : TON; (* On_Delay *)
    ON_Delay1 : TON; (* On_Delay *)
    P1O1A_FS : TON; (* P101A FS DELAY TIME *)
    P301A_Delay : TON;
    P301A_FS : TON;
    P301B_FS : TON;
    P301C : TON; (* initial values: P301C.Q=P301C RUN DELAY TIME *)
    P301C_FS : TON;
    P302A_FS : TON;
    P302B_FS : TON;
    P302C : TON; (* initial values: P302C.Q=P302C RUN DELAY TIME *)
    P302C_FS : TON;
    P303A_FS : TON;
    P303B_FS : TON;
    P303C : TON; (* initial values: P303C.Q=P302C RUN DELAY TIME *)
    P303C_FS : TON;
    P303_FS : TON;
    SINGLE_RUN_A : BOOL; (* A-SIDE 단독 런모드 *)
    SINGLE_RUN_B : BOOL; (* B-SIDE 단독 런 모드 *)
    T1 : TON; (* P301A-Trouble delay *)
    T10 : TON; (* P301C-3Min Stop delay *)
    T11 : TON; (* P302A Trouble-delay *)
    T12 : TON; (* P302B Trouble-delay *)
    T13 : TON; (* P302C-3Min Stop *)
    T14 : TON; (* P301C-3Min Stop delay *)
    T15 : TON; (* P301C-3Min Stop delay *)
    T2 : TON; (* P301B-Trouble delay *)
    T20 : TON; (* Reset *)
    T21 : TON; (* Reset *)
    T3 : TON; (* P301C-Trouble delay *)
    T301C : TON;
    T302C : TON; (* initial values: T302C.Q=P301C RUN DELAY TIME *)
    T4 : TON; (* P302A-Trouble delay *)
    T5 : TON; (* P302B-Trouble delay *)
    T6 : TIME; (* P302C-Trouble *)
    T6_사본1 : TON; (* P302C-Trouble delay *)
    T6_사본2 : TON; (* P302C-Trouble delay *)
    T7 : TON; (* P301C-3Min Stop delay *)
    T8 : TON; (* P301C-3Min Stop delay *)
    T9 : TON; (* P301C-3Min Stop delay *)
END_VAR
VAR_EXTERNAL
    _0100_CH5_DATA : INT; (* AT %UW1.0.7 *) (* 아날로그입력 모듈: 채널5 변환값 *)
END_VAR
VAR
    _e1 : R_TRIG;
    _e2 : R_TRIG;
END_VAR

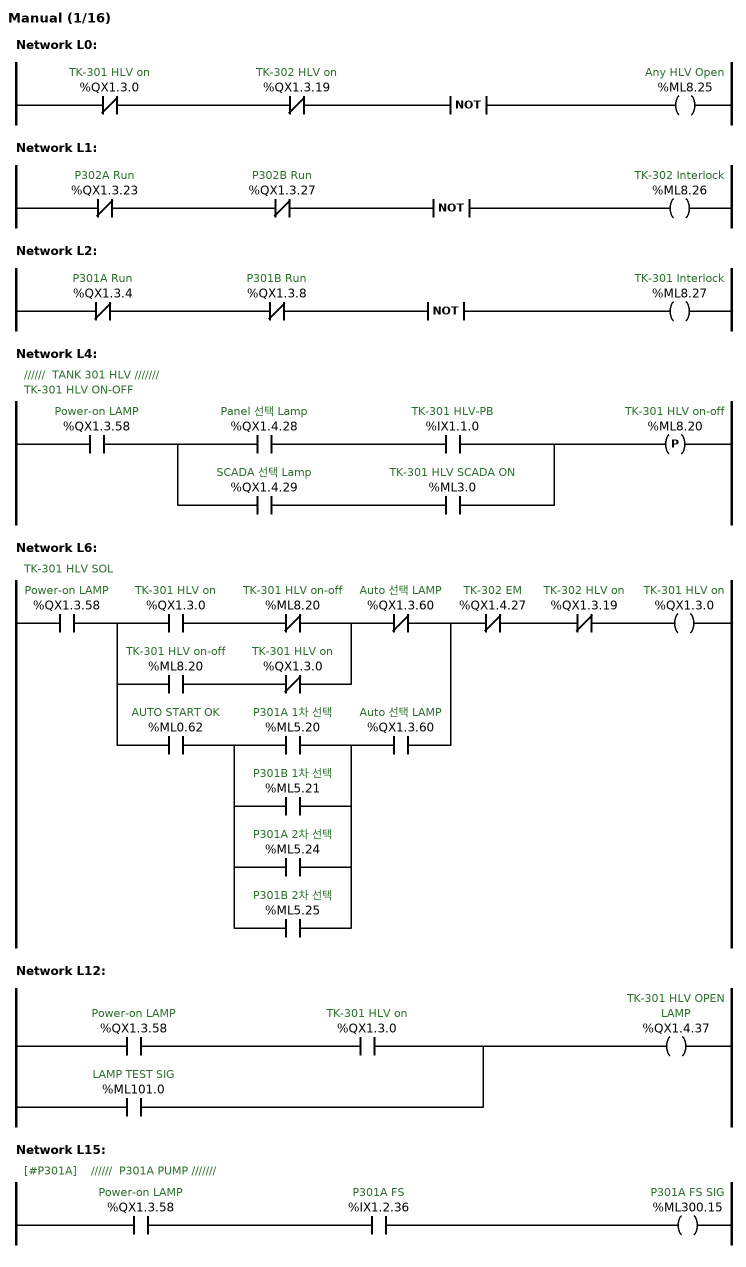
(* Rung L0 *)
%ML8.25 := NOT (NOT %QX1.3.0 AND NOT %QX1.3.19);
(* Rung L1 *)
%ML8.26 := NOT (NOT %QX1.3.23 AND NOT %QX1.3.27);
(* Rung L2 *)
%ML8.27 := NOT (NOT %QX1.3.4 AND NOT %QX1.3.8);
(* //////  TANK 301 HLV /////// *)
(* Rung L4 *)
_e1(CLK := %QX1.3.58 AND ((%QX1.4.28 AND %IX1.1.0) OR (%QX1.4.29 AND %ML3.0)));
%ML8.20 := _e1.Q;
(* TK-301 HLV ON-OFF *)
(* Rung L6 *)
%QX1.3.0 := %QX1.3.58 AND ((((%QX1.3.0 AND NOT %ML8.20) OR (%ML8.20 AND NOT %QX1.3.0)) AND NOT %QX1.3.60) OR (%ML0.62 AND (%ML5.20 OR %ML5.21 OR %ML5.24 OR %ML5.25) AND %QX1.3.60)) AND NOT %QX1.4.27 AND NOT %QX1.3.19;
(* TK-301 HLV SOL *)
(* Rung L12 *)
%QX1.4.37 := (%QX1.3.58 AND %QX1.3.0) OR %ML101.0;
(* [#P301A]    //////  P301A PUMP /////// *)
(* Rung L15 *)
%ML300.15 := %QX1.3.58 AND %IX1.2.36;

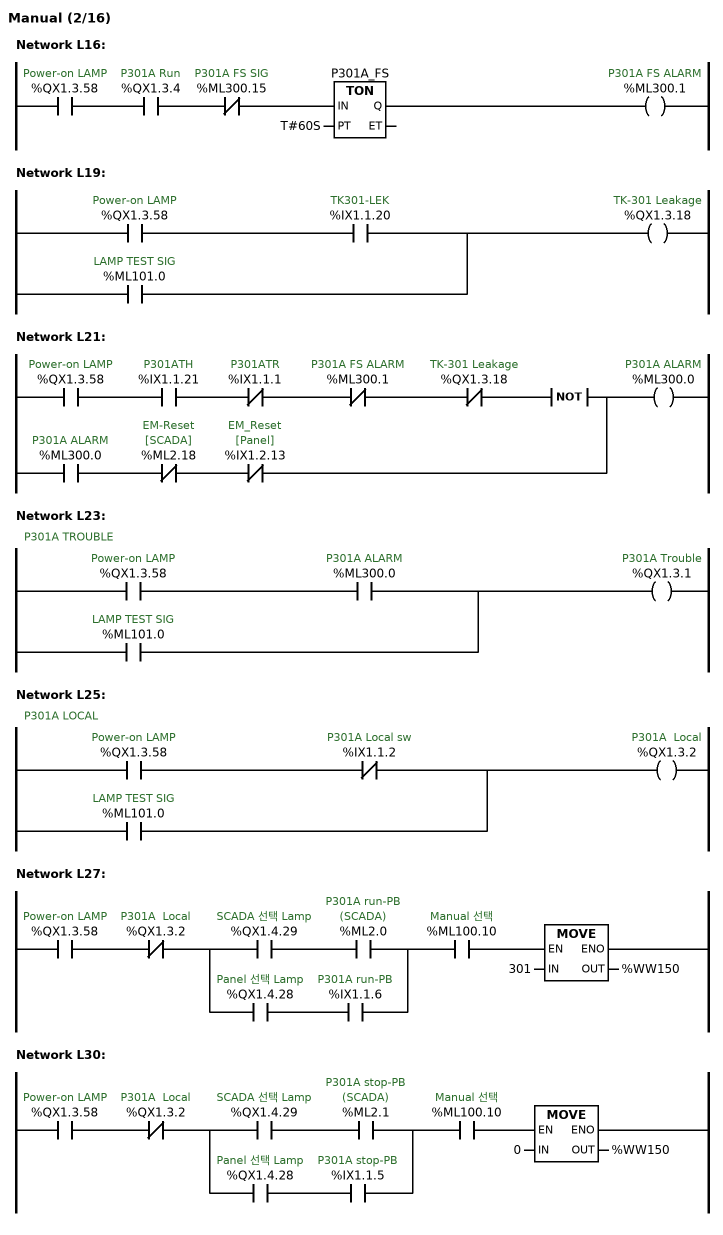
(* Rung L16 *)
P301A_FS(IN := %QX1.3.58 AND %QX1.3.4 AND NOT %ML300.15, PT := T#60S);
%ML300.1 := P301A_FS.Q;
(* Rung L19 *)
%QX1.3.18 := (%QX1.3.58 AND %IX1.1.20) OR %ML101.0;
(* Rung L21 *)
%ML300.0 := NOT (%QX1.3.58 AND %IX1.1.21 AND NOT %IX1.1.1 AND NOT %ML300.1 AND NOT %QX1.3.18) OR (%ML300.0 AND NOT %ML2.18 AND NOT %IX1.2.13);
(* Rung L23 *)
%QX1.3.1 := (%QX1.3.58 AND %ML300.0) OR %ML101.0;
(* P301A TROUBLE *)
(* Rung L25 *)
%QX1.3.2 := (%QX1.3.58 AND NOT %IX1.1.2) OR %ML101.0;
(* P301A LOCAL *)
(* Rung L27 *)
IF %QX1.3.58 AND NOT %QX1.3.2 AND ((%QX1.4.29 AND %ML2.0) OR (%QX1.4.28 AND %IX1.1.6)) AND %ML100.10 THEN
    %WW150 := 301;
END_IF;
(* Rung L30 *)
IF %QX1.3.58 AND NOT %QX1.3.2 AND ((%QX1.4.29 AND %ML2.1) OR (%QX1.4.28 AND %IX1.1.5)) AND %ML100.10 THEN
    %WW150 := 0;
END_IF;

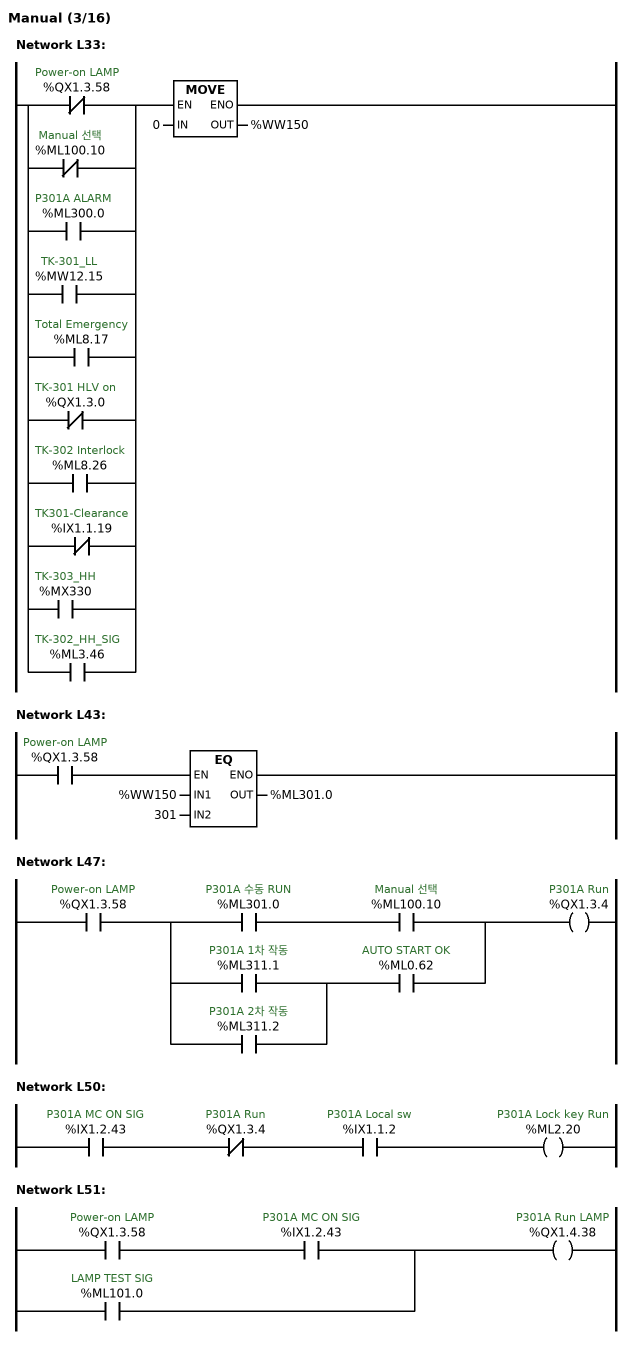
(* Rung L33 *)
IF NOT %QX1.3.58 OR NOT %ML100.10 OR %ML300.0 OR %MW12.15 OR %ML8.17 OR NOT %QX1.3.0 OR %ML8.26 OR NOT %IX1.1.19 OR %MX330 OR %ML3.46 THEN
    %WW150 := 0;
END_IF;
(* Rung L43 *)
IF %QX1.3.58 THEN %ML301.0 := %WW150 = 301; END_IF;
(* Rung L47 *)
%QX1.3.4 := %QX1.3.58 AND ((%ML301.0 AND %ML100.10) OR ((%ML311.1 OR %ML311.2) AND %ML0.62));
(* Rung L50 *)
%ML2.20 := %IX1.2.43 AND NOT %QX1.3.4 AND %IX1.1.2;
(* Rung L51 *)
%QX1.4.38 := (%QX1.3.58 AND %IX1.2.43) OR %ML101.0;

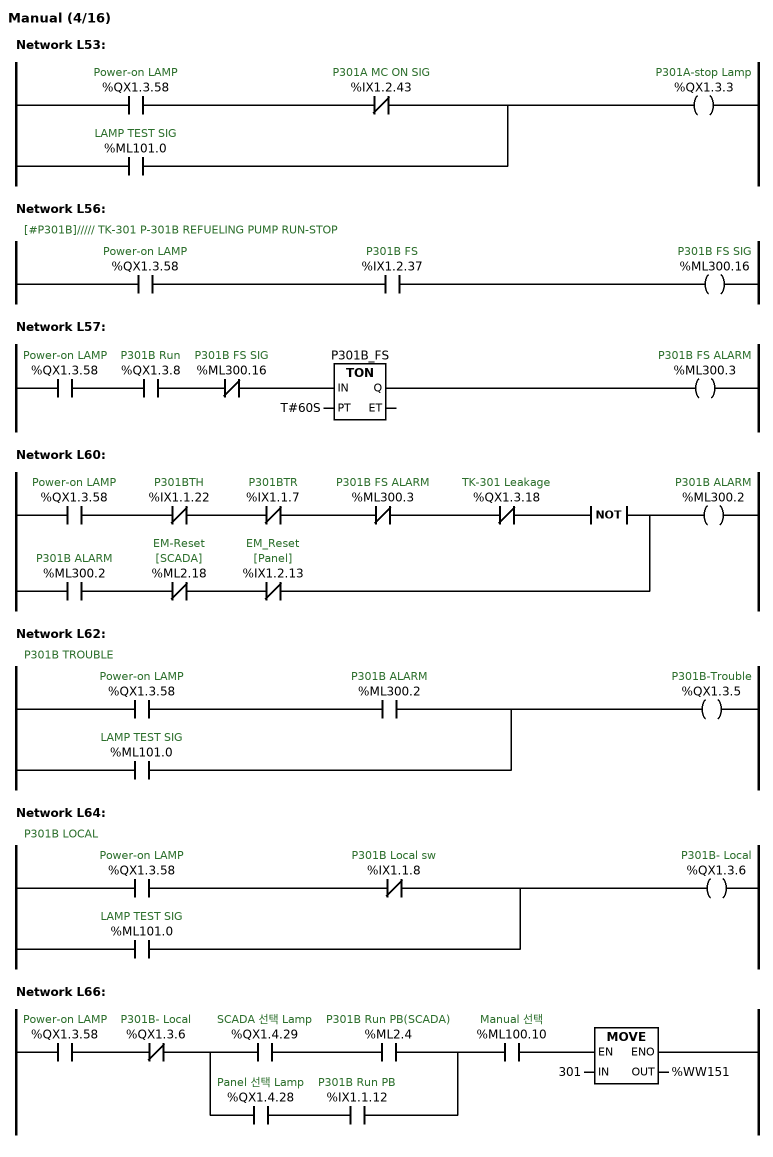
(* Rung L53 *)
%QX1.3.3 := (%QX1.3.58 AND NOT %IX1.2.43) OR %ML101.0;
(* [#P301B]///// TK-301 P-301B REFUELING PUMP RUN-STOP *)
(* Rung L56 *)
%ML300.16 := %QX1.3.58 AND %IX1.2.37;
(* Rung L57 *)
P301B_FS(IN := %QX1.3.58 AND %QX1.3.8 AND NOT %ML300.16, PT := T#60S);
%ML300.3 := P301B_FS.Q;
(* Rung L60 *)
%ML300.2 := NOT (%QX1.3.58 AND NOT %IX1.1.22 AND NOT %IX1.1.7 AND NOT %ML300.3 AND NOT %QX1.3.18) OR (%ML300.2 AND NOT %ML2.18 AND NOT %IX1.2.13);
(* Rung L62 *)
%QX1.3.5 := (%QX1.3.58 AND %ML300.2) OR %ML101.0;
(* P301B TROUBLE *)
(* Rung L64 *)
%QX1.3.6 := (%QX1.3.58 AND NOT %IX1.1.8) OR %ML101.0;
(* P301B LOCAL *)
(* Rung L66 *)
IF %QX1.3.58 AND NOT %QX1.3.6 AND ((%QX1.4.29 AND %ML2.4) OR (%QX1.4.28 AND %IX1.1.12)) AND %ML100.10 THEN
    %WW151 := 301;
END_IF;

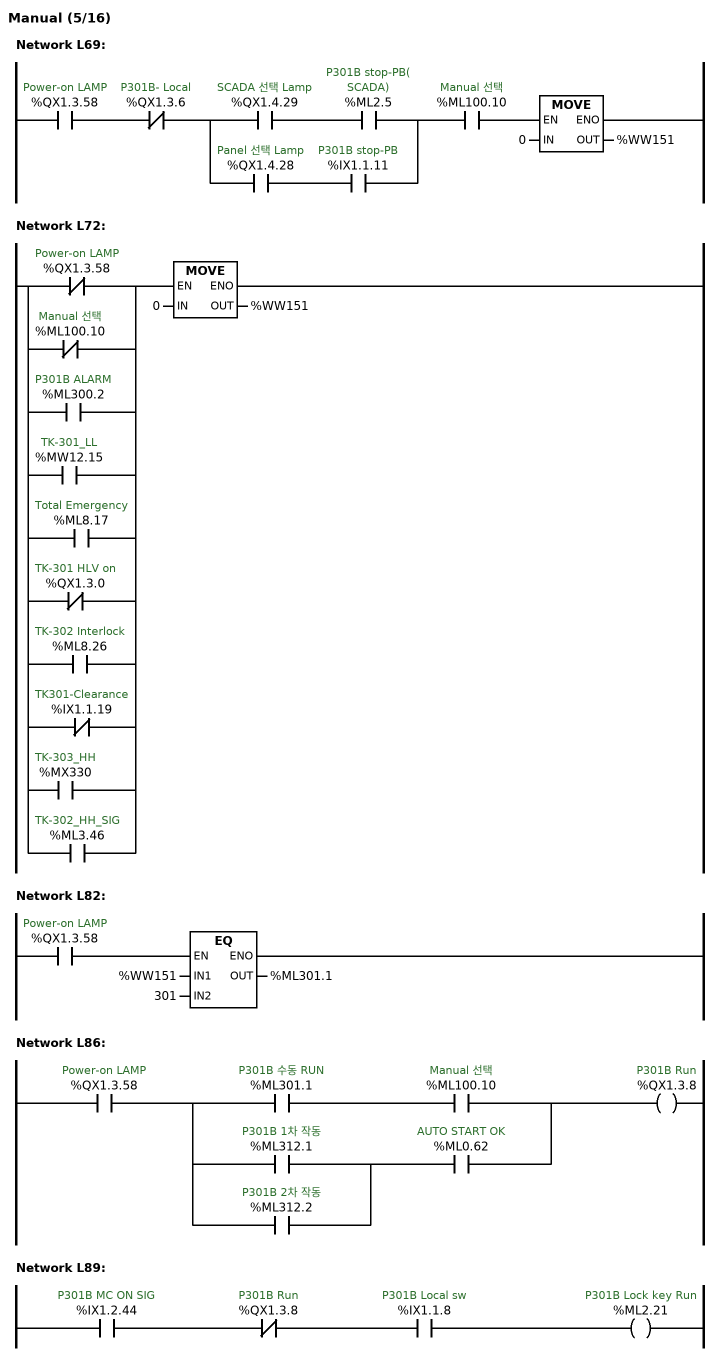
(* Rung L69 *)
IF %QX1.3.58 AND NOT %QX1.3.6 AND ((%QX1.4.29 AND %ML2.5) OR (%QX1.4.28 AND %IX1.1.11)) AND %ML100.10 THEN
    %WW151 := 0;
END_IF;
(* Rung L72 *)
IF NOT %QX1.3.58 OR NOT %ML100.10 OR %ML300.2 OR %MW12.15 OR %ML8.17 OR NOT %QX1.3.0 OR %ML8.26 OR NOT %IX1.1.19 OR %MX330 OR %ML3.46 THEN
    %WW151 := 0;
END_IF;
(* Rung L82 *)
IF %QX1.3.58 THEN %ML301.1 := %WW151 = 301; END_IF;
(* Rung L86 *)
%QX1.3.8 := %QX1.3.58 AND ((%ML301.1 AND %ML100.10) OR ((%ML312.1 OR %ML312.2) AND %ML0.62));
(* Rung L89 *)
%ML2.21 := %IX1.2.44 AND NOT %QX1.3.8 AND %IX1.1.8;

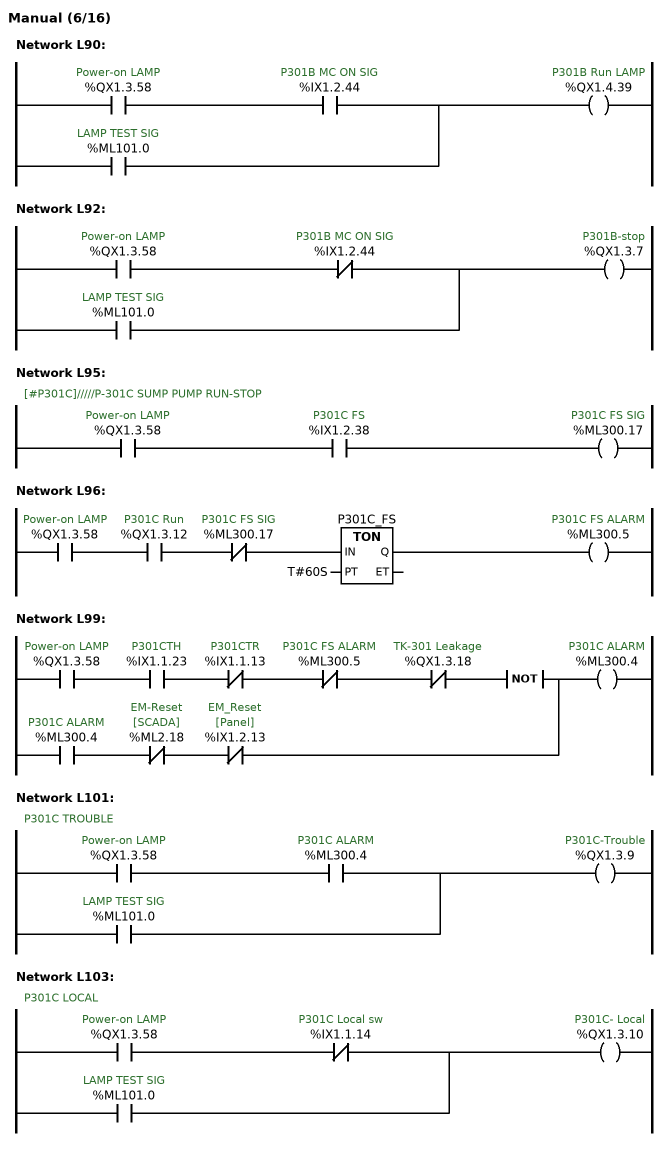
(* Rung L90 *)
%QX1.4.39 := (%QX1.3.58 AND %IX1.2.44) OR %ML101.0;
(* Rung L92 *)
%QX1.3.7 := (%QX1.3.58 AND NOT %IX1.2.44) OR %ML101.0;
(* [#P301C]/////P-301C SUMP PUMP RUN-STOP *)
(* Rung L95 *)
%ML300.17 := %QX1.3.58 AND %IX1.2.38;
(* Rung L96 *)
P301C_FS(IN := %QX1.3.58 AND %QX1.3.12 AND NOT %ML300.17, PT := T#60S);
%ML300.5 := P301C_FS.Q;
(* Rung L99 *)
%ML300.4 := NOT (%QX1.3.58 AND %IX1.1.23 AND NOT %IX1.1.13 AND NOT %ML300.5 AND NOT %QX1.3.18) OR (%ML300.4 AND NOT %ML2.18 AND NOT %IX1.2.13);
(* Rung L101 *)
%QX1.3.9 := (%QX1.3.58 AND %ML300.4) OR %ML101.0;
(* P301C TROUBLE *)
(* Rung L103 *)
%QX1.3.10 := (%QX1.3.58 AND NOT %IX1.1.14) OR %ML101.0;
(* P301C LOCAL *)

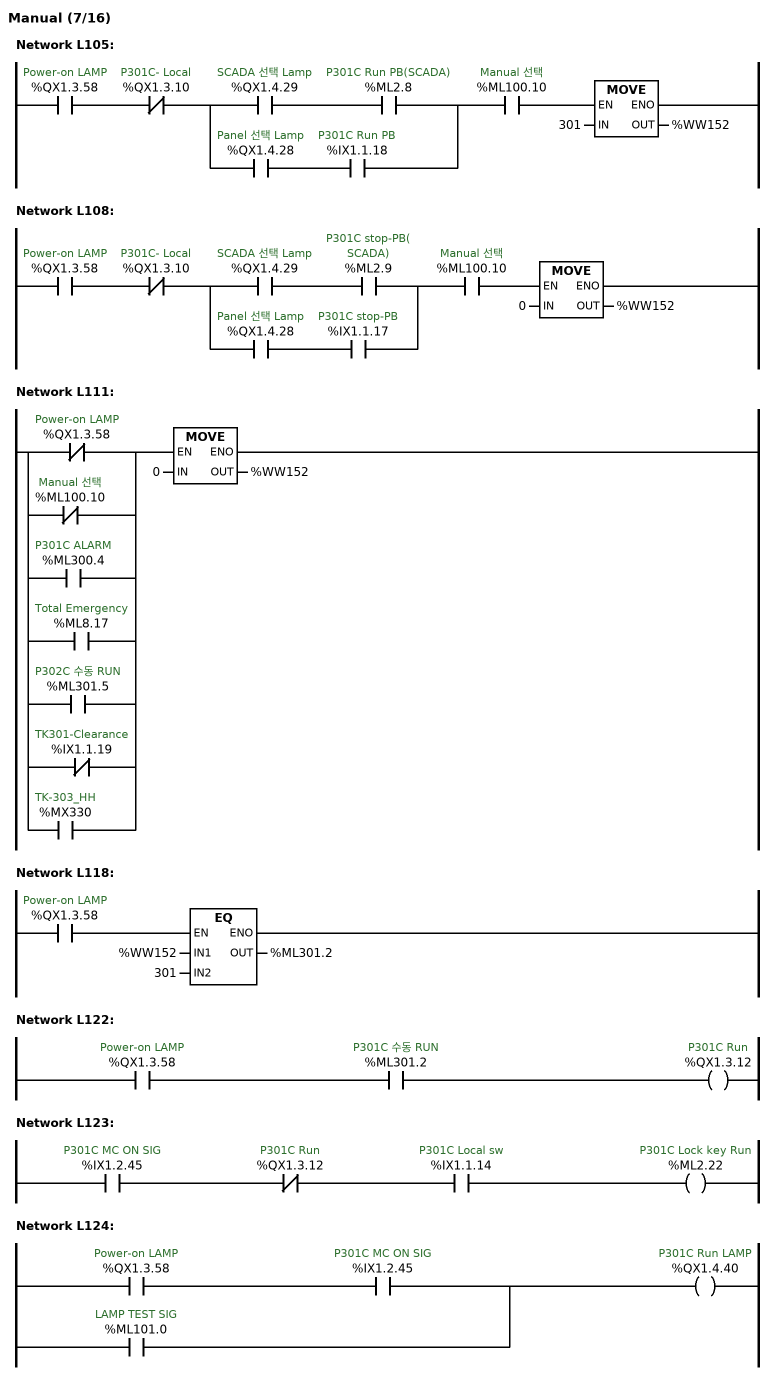
(* Rung L105 *)
IF %QX1.3.58 AND NOT %QX1.3.10 AND ((%QX1.4.29 AND %ML2.8) OR (%QX1.4.28 AND %IX1.1.18)) AND %ML100.10 THEN
    %WW152 := 301;
END_IF;
(* Rung L108 *)
IF %QX1.3.58 AND NOT %QX1.3.10 AND ((%QX1.4.29 AND %ML2.9) OR (%QX1.4.28 AND %IX1.1.17)) AND %ML100.10 THEN
    %WW152 := 0;
END_IF;
(* Rung L111 *)
IF NOT %QX1.3.58 OR NOT %ML100.10 OR %ML300.4 OR %ML8.17 OR %ML301.5 OR NOT %IX1.1.19 OR %MX330 THEN
    %WW152 := 0;
END_IF;
(* Rung L118 *)
IF %QX1.3.58 THEN %ML301.2 := %WW152 = 301; END_IF;
(* Rung L122 *)
%QX1.3.12 := %QX1.3.58 AND %ML301.2;
(* Rung L123 *)
%ML2.22 := %IX1.2.45 AND NOT %QX1.3.12 AND %IX1.1.14;
(* Rung L124 *)
%QX1.4.40 := (%QX1.3.58 AND %IX1.2.45) OR %ML101.0;

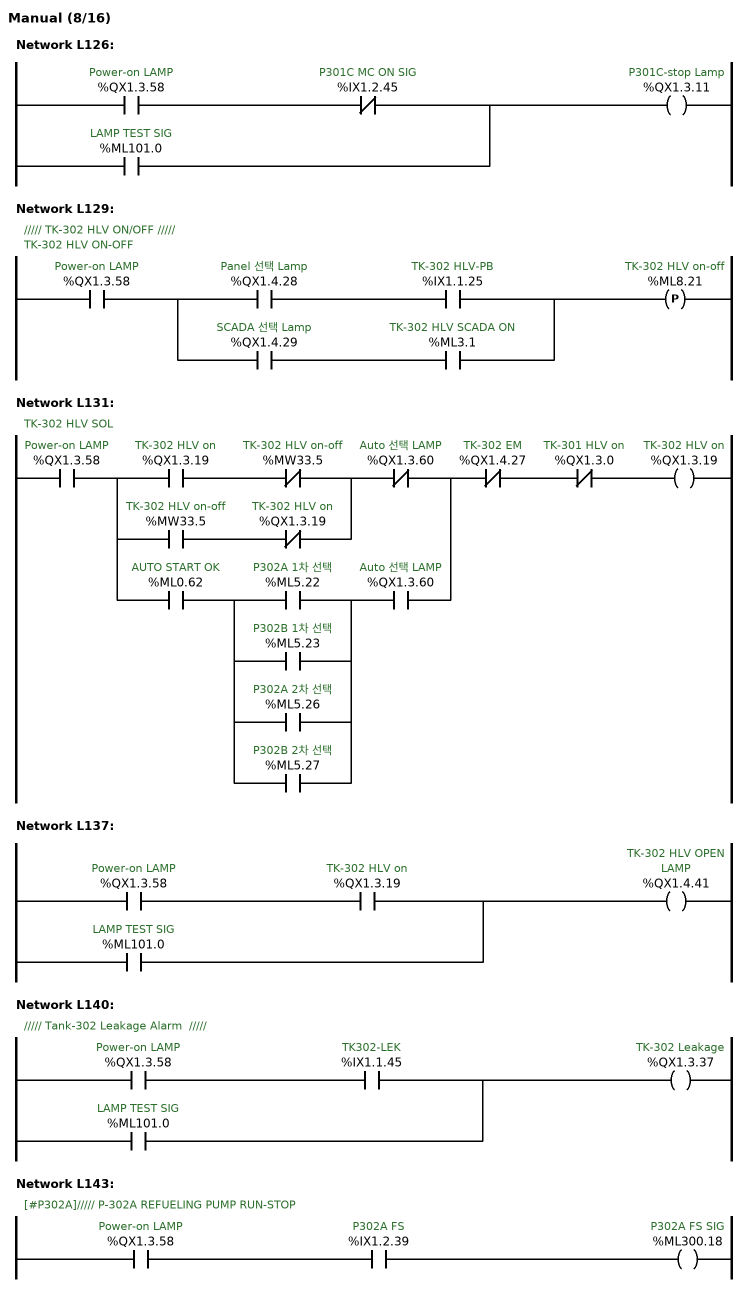
(* Rung L126 *)
%QX1.3.11 := (%QX1.3.58 AND NOT %IX1.2.45) OR %ML101.0;
(* ///// TK-302 HLV ON/OFF ///// *)
(* Rung L129 *)
_e2(CLK := %QX1.3.58 AND ((%QX1.4.28 AND %IX1.1.25) OR (%QX1.4.29 AND %ML3.1)));
%ML8.21 := _e2.Q;
(* TK-302 HLV ON-OFF *)
(* Rung L131 *)
%QX1.3.19 := %QX1.3.58 AND ((((%QX1.3.19 AND NOT %MW33.5) OR (%MW33.5 AND NOT %QX1.3.19)) AND NOT %QX1.3.60) OR (%ML0.62 AND (%ML5.22 OR %ML5.23 OR %ML5.26 OR %ML5.27) AND %QX1.3.60)) AND NOT %QX1.4.27 AND NOT %QX1.3.0;
(* TK-302 HLV SOL *)
(* Rung L137 *)
%QX1.4.41 := (%QX1.3.58 AND %QX1.3.19) OR %ML101.0;
(* ///// Tank-302 Leakage Alarm  ///// *)
(* Rung L140 *)
%QX1.3.37 := (%QX1.3.58 AND %IX1.1.45) OR %ML101.0;
(* [#P302A]///// P-302A REFUELING PUMP RUN-STOP *)
(* Rung L143 *)
%ML300.18 := %QX1.3.58 AND %IX1.2.39;

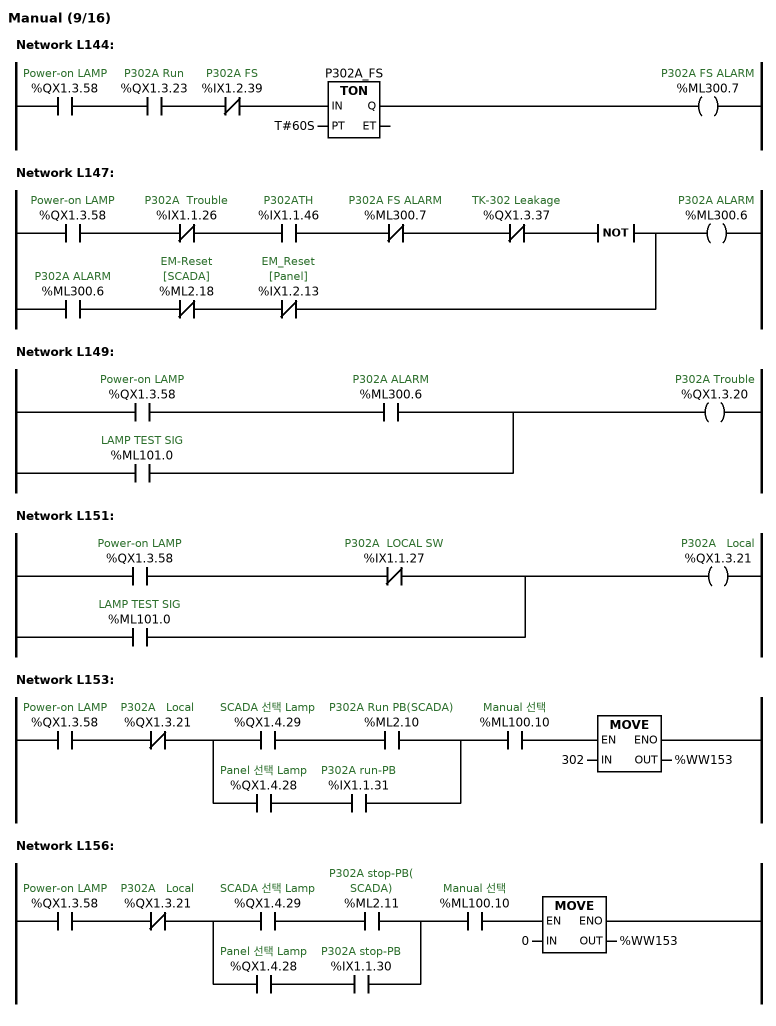
(* Rung L144 *)
P302A_FS(IN := %QX1.3.58 AND %QX1.3.23 AND NOT %IX1.2.39, PT := T#60S);
%ML300.7 := P302A_FS.Q;
(* Rung L147 *)
%ML300.6 := NOT (%QX1.3.58 AND NOT %IX1.1.26 AND %IX1.1.46 AND NOT %ML300.7 AND NOT %QX1.3.37) OR (%ML300.6 AND NOT %ML2.18 AND NOT %IX1.2.13);
(* Rung L149 *)
%QX1.3.20 := (%QX1.3.58 AND %ML300.6) OR %ML101.0;
(* Rung L151 *)
%QX1.3.21 := (%QX1.3.58 AND NOT %IX1.1.27) OR %ML101.0;
(* Rung L153 *)
IF %QX1.3.58 AND NOT %QX1.3.21 AND ((%QX1.4.29 AND %ML2.10) OR (%QX1.4.28 AND %IX1.1.31)) AND %ML100.10 THEN
    %WW153 := 302;
END_IF;
(* Rung L156 *)
IF %QX1.3.58 AND NOT %QX1.3.21 AND ((%QX1.4.29 AND %ML2.11) OR (%QX1.4.28 AND %IX1.1.30)) AND %ML100.10 THEN
    %WW153 := 0;
END_IF;

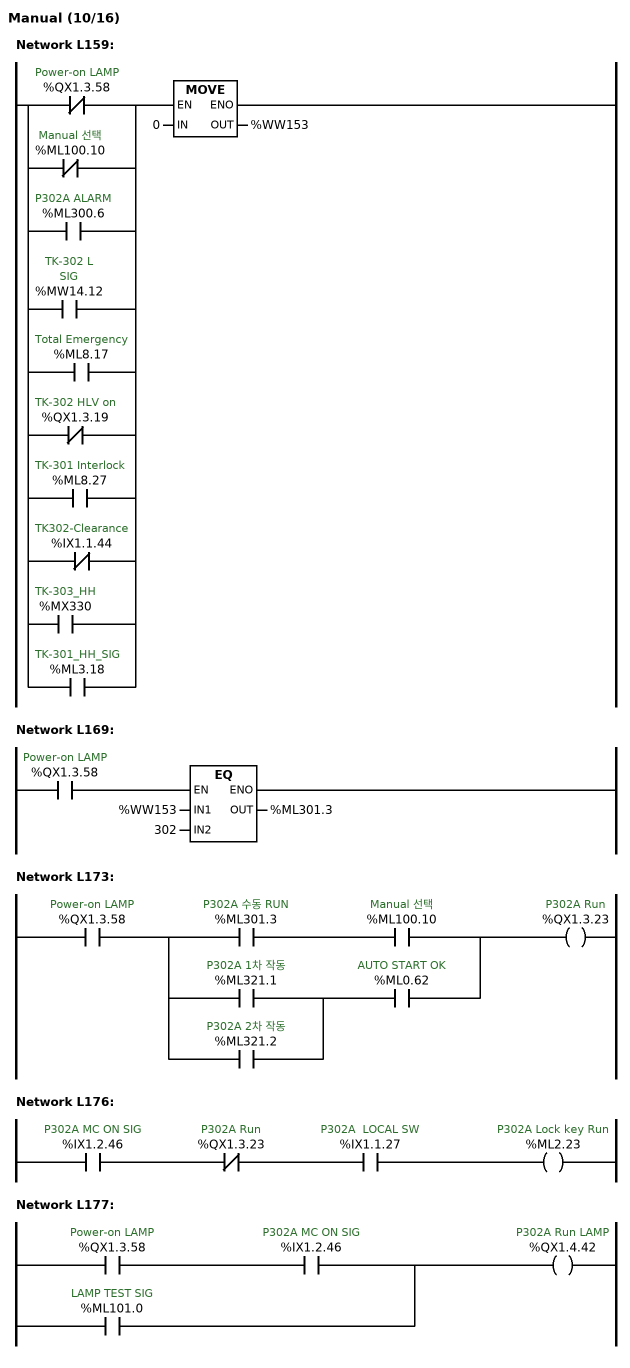
(* Rung L159 *)
IF NOT %QX1.3.58 OR NOT %ML100.10 OR %ML300.6 OR %MW14.12 OR %ML8.17 OR NOT %QX1.3.19 OR %ML8.27 OR NOT %IX1.1.44 OR %MX330 OR %ML3.18 THEN
    %WW153 := 0;
END_IF;
(* Rung L169 *)
IF %QX1.3.58 THEN %ML301.3 := %WW153 = 302; END_IF;
(* Rung L173 *)
%QX1.3.23 := %QX1.3.58 AND ((%ML301.3 AND %ML100.10) OR ((%ML321.1 OR %ML321.2) AND %ML0.62));
(* Rung L176 *)
%ML2.23 := %IX1.2.46 AND NOT %QX1.3.23 AND %IX1.1.27;
(* Rung L177 *)
%QX1.4.42 := (%QX1.3.58 AND %IX1.2.46) OR %ML101.0;

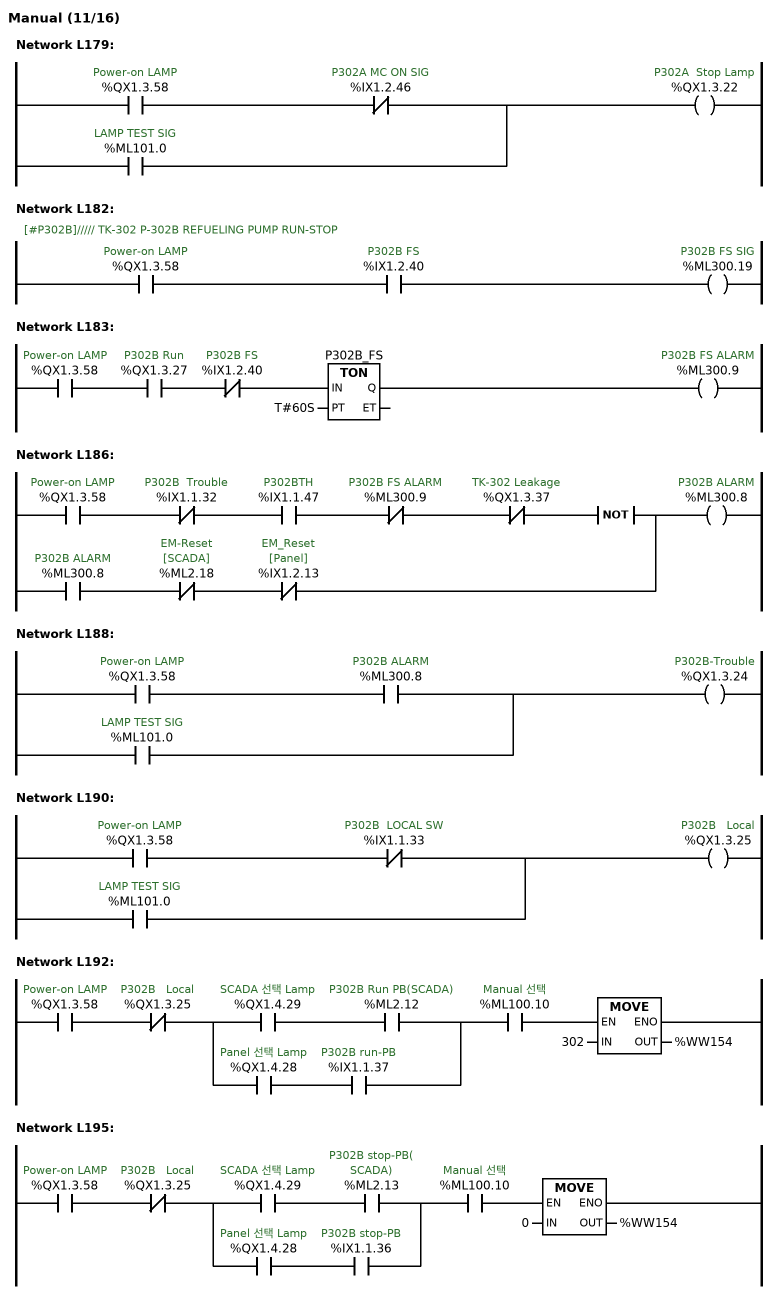
(* Rung L179 *)
%QX1.3.22 := (%QX1.3.58 AND NOT %IX1.2.46) OR %ML101.0;
(* [#P302B]///// TK-302 P-302B REFUELING PUMP RUN-STOP *)
(* Rung L182 *)
%ML300.19 := %QX1.3.58 AND %IX1.2.40;
(* Rung L183 *)
P302B_FS(IN := %QX1.3.58 AND %QX1.3.27 AND NOT %IX1.2.40, PT := T#60S);
%ML300.9 := P302B_FS.Q;
(* Rung L186 *)
%ML300.8 := NOT (%QX1.3.58 AND NOT %IX1.1.32 AND %IX1.1.47 AND NOT %ML300.9 AND NOT %QX1.3.37) OR (%ML300.8 AND NOT %ML2.18 AND NOT %IX1.2.13);
(* Rung L188 *)
%QX1.3.24 := (%QX1.3.58 AND %ML300.8) OR %ML101.0;
(* Rung L190 *)
%QX1.3.25 := (%QX1.3.58 AND NOT %IX1.1.33) OR %ML101.0;
(* Rung L192 *)
IF %QX1.3.58 AND NOT %QX1.3.25 AND ((%QX1.4.29 AND %ML2.12) OR (%QX1.4.28 AND %IX1.1.37)) AND %ML100.10 THEN
    %WW154 := 302;
END_IF;
(* Rung L195 *)
IF %QX1.3.58 AND NOT %QX1.3.25 AND ((%QX1.4.29 AND %ML2.13) OR (%QX1.4.28 AND %IX1.1.36)) AND %ML100.10 THEN
    %WW154 := 0;
END_IF;

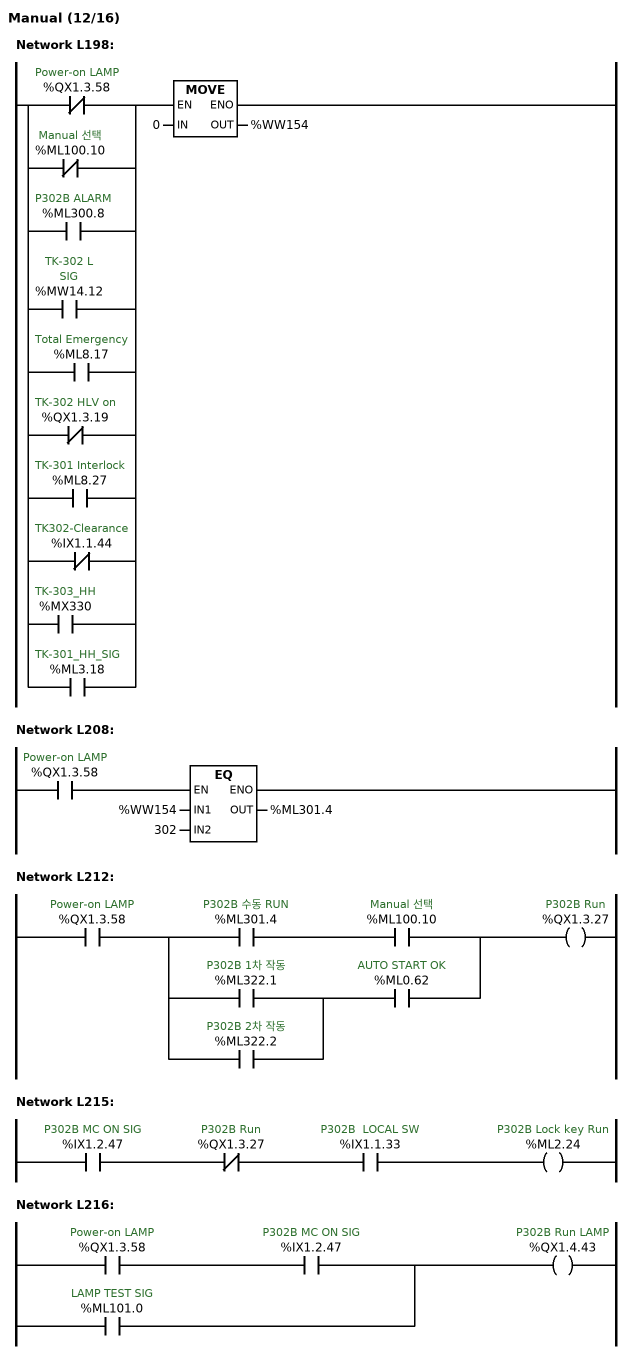
(* Rung L198 *)
IF NOT %QX1.3.58 OR NOT %ML100.10 OR %ML300.8 OR %MW14.12 OR %ML8.17 OR NOT %QX1.3.19 OR %ML8.27 OR NOT %IX1.1.44 OR %MX330 OR %ML3.18 THEN
    %WW154 := 0;
END_IF;
(* Rung L208 *)
IF %QX1.3.58 THEN %ML301.4 := %WW154 = 302; END_IF;
(* Rung L212 *)
%QX1.3.27 := %QX1.3.58 AND ((%ML301.4 AND %ML100.10) OR ((%ML322.1 OR %ML322.2) AND %ML0.62));
(* Rung L215 *)
%ML2.24 := %IX1.2.47 AND NOT %QX1.3.27 AND %IX1.1.33;
(* Rung L216 *)
%QX1.4.43 := (%QX1.3.58 AND %IX1.2.47) OR %ML101.0;

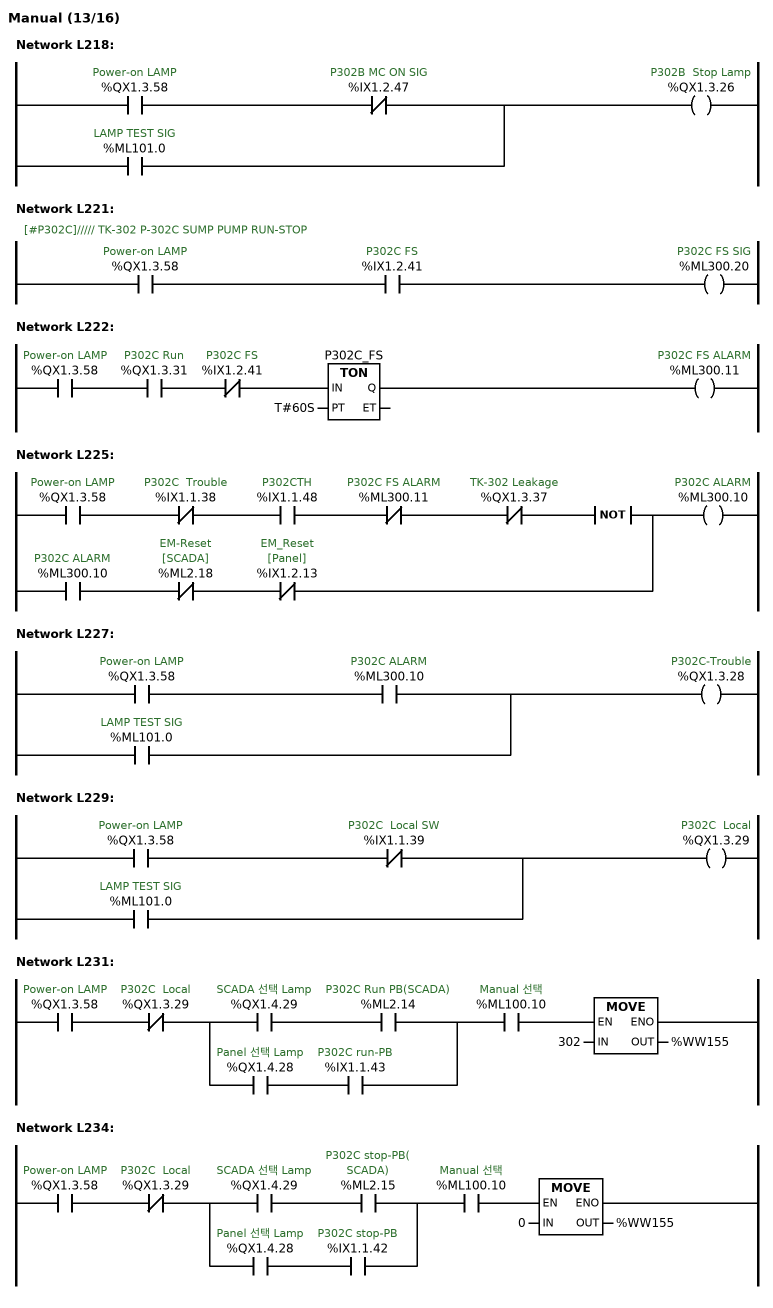
(* Rung L218 *)
%QX1.3.26 := (%QX1.3.58 AND NOT %IX1.2.47) OR %ML101.0;
(* [#P302C]///// TK-302 P-302C SUMP PUMP RUN-STOP *)
(* Rung L221 *)
%ML300.20 := %QX1.3.58 AND %IX1.2.41;
(* Rung L222 *)
P302C_FS(IN := %QX1.3.58 AND %QX1.3.31 AND NOT %IX1.2.41, PT := T#60S);
%ML300.11 := P302C_FS.Q;
(* Rung L225 *)
%ML300.10 := NOT (%QX1.3.58 AND NOT %IX1.1.38 AND %IX1.1.48 AND NOT %ML300.11 AND NOT %QX1.3.37) OR (%ML300.10 AND NOT %ML2.18 AND NOT %IX1.2.13);
(* Rung L227 *)
%QX1.3.28 := (%QX1.3.58 AND %ML300.10) OR %ML101.0;
(* Rung L229 *)
%QX1.3.29 := (%QX1.3.58 AND NOT %IX1.1.39) OR %ML101.0;
(* Rung L231 *)
IF %QX1.3.58 AND NOT %QX1.3.29 AND ((%QX1.4.29 AND %ML2.14) OR (%QX1.4.28 AND %IX1.1.43)) AND %ML100.10 THEN
    %WW155 := 302;
END_IF;
(* Rung L234 *)
IF %QX1.3.58 AND NOT %QX1.3.29 AND ((%QX1.4.29 AND %ML2.15) OR (%QX1.4.28 AND %IX1.1.42)) AND %ML100.10 THEN
    %WW155 := 0;
END_IF;

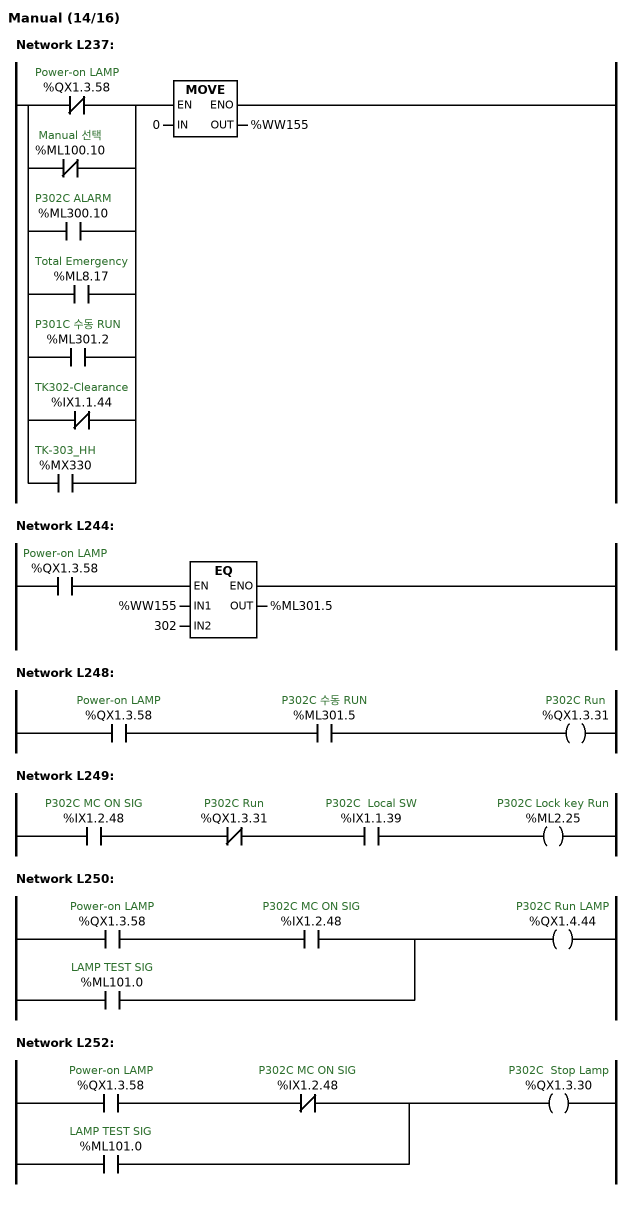
(* Rung L237 *)
IF NOT %QX1.3.58 OR NOT %ML100.10 OR %ML300.10 OR %ML8.17 OR %ML301.2 OR NOT %IX1.1.44 OR %MX330 THEN
    %WW155 := 0;
END_IF;
(* Rung L244 *)
IF %QX1.3.58 THEN %ML301.5 := %WW155 = 302; END_IF;
(* Rung L248 *)
%QX1.3.31 := %QX1.3.58 AND %ML301.5;
(* Rung L249 *)
%ML2.25 := %IX1.2.48 AND NOT %QX1.3.31 AND %IX1.1.39;
(* Rung L250 *)
%QX1.4.44 := (%QX1.3.58 AND %IX1.2.48) OR %ML101.0;
(* Rung L252 *)
%QX1.3.30 := (%QX1.3.58 AND NOT %IX1.2.48) OR %ML101.0;

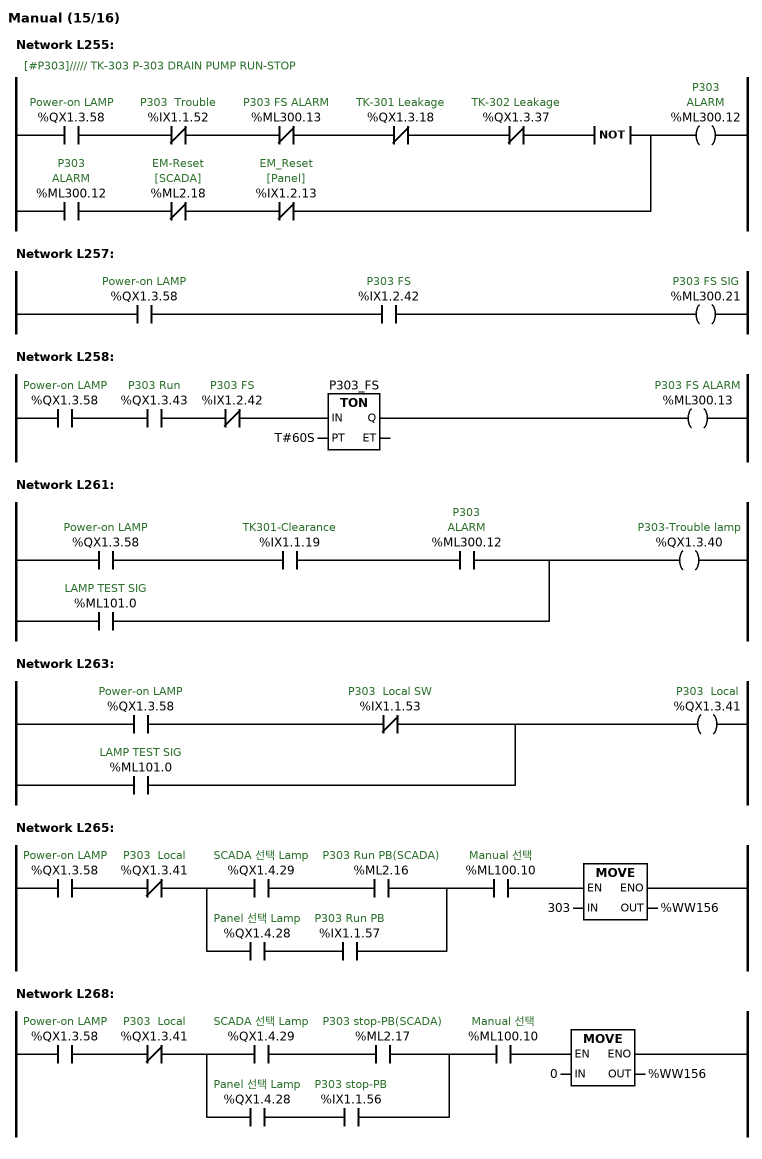
(* [#P303]///// TK-303 P-303 DRAIN PUMP RUN-STOP *)
(* Rung L255 *)
%ML300.12 := NOT (%QX1.3.58 AND NOT %IX1.1.52 AND NOT %ML300.13 AND NOT %QX1.3.18 AND NOT %QX1.3.37) OR (%ML300.12 AND NOT %ML2.18 AND NOT %IX1.2.13);
(* Rung L257 *)
%ML300.21 := %QX1.3.58 AND %IX1.2.42;
(* Rung L258 *)
P303_FS(IN := %QX1.3.58 AND %QX1.3.43 AND NOT %IX1.2.42, PT := T#60S);
%ML300.13 := P303_FS.Q;
(* Rung L261 *)
%QX1.3.40 := (%QX1.3.58 AND %IX1.1.19 AND %ML300.12) OR %ML101.0;
(* Rung L263 *)
%QX1.3.41 := (%QX1.3.58 AND NOT %IX1.1.53) OR %ML101.0;
(* Rung L265 *)
IF %QX1.3.58 AND NOT %QX1.3.41 AND ((%QX1.4.29 AND %ML2.16) OR (%QX1.4.28 AND %IX1.1.57)) AND %ML100.10 THEN
    %WW156 := 303;
END_IF;
(* Rung L268 *)
IF %QX1.3.58 AND NOT %QX1.3.41 AND ((%QX1.4.29 AND %ML2.17) OR (%QX1.4.28 AND %IX1.1.56)) AND %ML100.10 THEN
    %WW156 := 0;
END_IF;

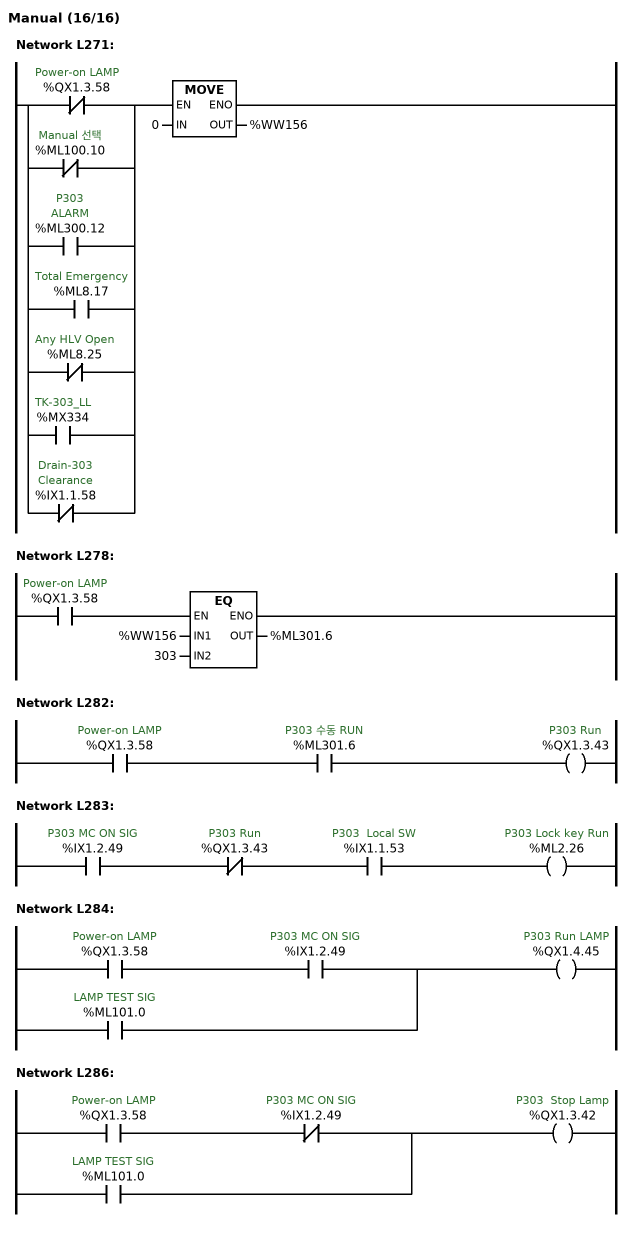
(* Rung L271 *)
IF NOT %QX1.3.58 OR NOT %ML100.10 OR %ML300.12 OR %ML8.17 OR NOT %ML8.25 OR %MX334 OR NOT %IX1.1.58 THEN
    %WW156 := 0;
END_IF;
(* Rung L278 *)
IF %QX1.3.58 THEN %ML301.6 := %WW156 = 303; END_IF;
(* Rung L282 *)
%QX1.3.43 := %QX1.3.58 AND %ML301.6;
(* Rung L283 *)
%ML2.26 := %IX1.2.49 AND NOT %QX1.3.43 AND %IX1.1.53;
(* Rung L284 *)
%QX1.4.45 := (%QX1.3.58 AND %IX1.2.49) OR %ML101.0;
(* Rung L286 *)
%QX1.3.42 := (%QX1.3.58 AND NOT %IX1.2.49) OR %ML101.0;
END_PROGRAM

PROGRAM Automatic (* task: 스캔 프로그램 *)
VAR
    AUTO_STR : TON;
    INST : TON;
    one_set_run : TON;
    one_set_run1 : TON;
    T34 : TON; (* 2차펌프 운전지연 *)
    T35 : TON; (* 2차정지 지연20S *)
    T36 : TON; (* 1차펌프 정지지연20S *)
    T37 : TON; (* Reset_Delay *)
    T38 : TON; (* Reset_초기화 *)
    T39 : TON; (* 2차정지 지연20S *)
    T40 : TON; (* 2차펌프 운전지연 *)
    T41 : TON; (* 2차정지 지연20S *)
    T42 : TON; (* 1차펌프 정지지연20S *)
    T43 : TON; (* Reset_초기화 *)
    T44 : TON; (* Reset_초기화 *)
    Two_set_run2 : TON;
    Two_set_stp : TON;
    Two_set_stp10 : TON;
    Two_set_stp11 : TON;
    Two_set_stp12 : TON;
    Two_set_stp2 : TON;
    Two_set_stp3 : TON;
    Two_set_stp4 : TON;
    Two_set_stp5 : TON;
    Two_set_stp6 : TON;
    Two_set_stp7 : TON;
    Two_set_stp8 : TON;
    Two_set_stp9 : TON;
END_VAR
VAR
    _p1 : BOOL;
    _p2 : BOOL;
    _t3 : BOOL;
    _t4 : BOOL;
    _t5 : DINT;
END_VAR

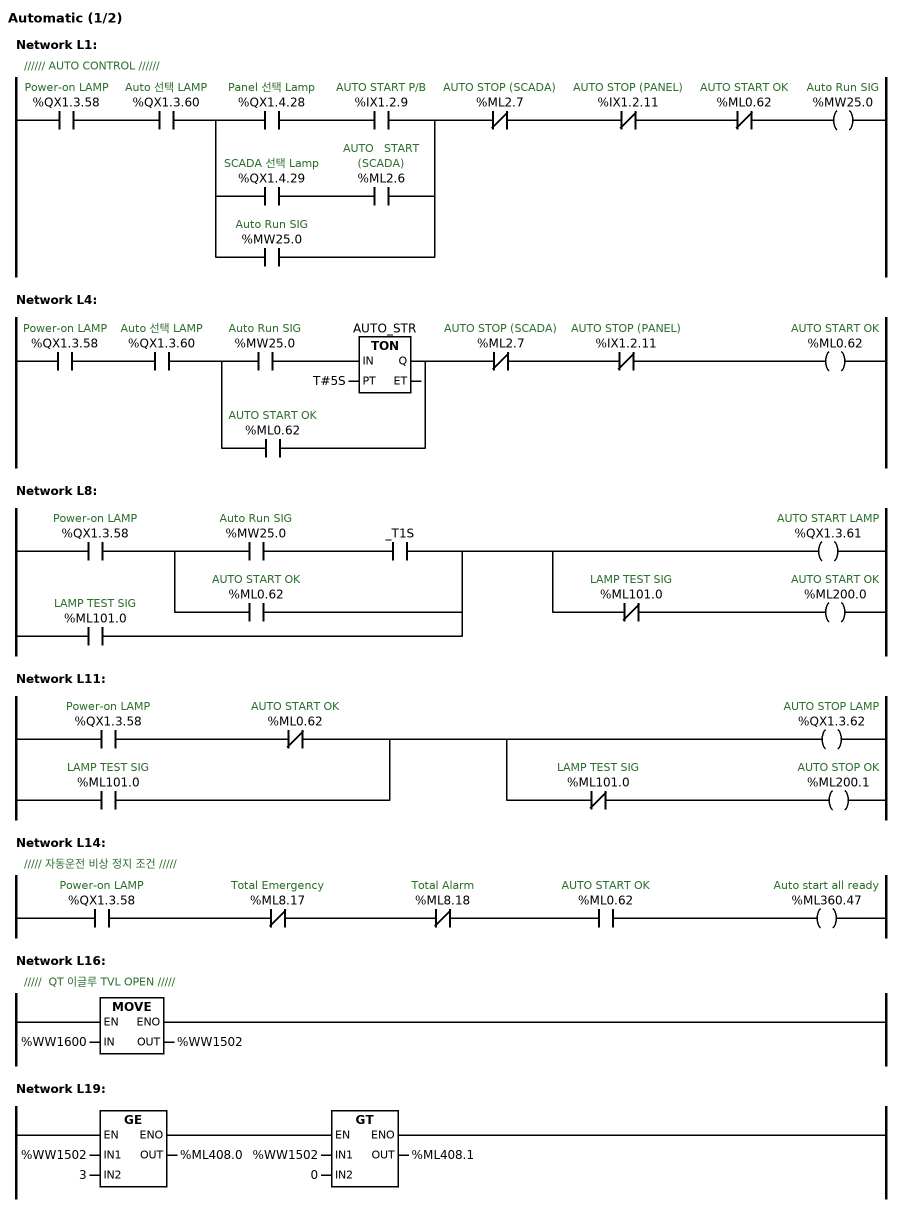
(* ////// AUTO CONTROL ////// *)
(* Rung L1 *)
%MW25.0 := %QX1.3.58 AND %QX1.3.60 AND ((%QX1.4.28 AND %IX1.2.9) OR (%QX1.4.29 AND %ML2.6) OR %MW25.0) AND NOT %ML2.7 AND NOT %IX1.2.11 AND NOT %ML0.62;
(* Rung L4 *)
AUTO_STR(IN := %QX1.3.58 AND %QX1.3.60 AND %MW25.0, PT := T#5S);
%ML0.62 := (AUTO_STR.Q OR (%QX1.3.58 AND %QX1.3.60 AND %ML0.62)) AND NOT %ML2.7 AND NOT %IX1.2.11;
(* Rung L8 *)
_p1 := (%QX1.3.58 AND ((%MW25.0 AND _T1S) OR %ML0.62)) OR %ML101.0;
%QX1.3.61 := _p1;
%ML200.0 := _p1 AND NOT %ML101.0;
(* Rung L11 *)
_p2 := (%QX1.3.58 AND NOT %ML0.62) OR %ML101.0;
%QX1.3.62 := _p2;
%ML200.1 := _p2 AND NOT %ML101.0;
(* ///// 자동운전 비상 정지 조건 ///// *)
(* Rung L14 *)
%ML360.47 := %QX1.3.58 AND NOT %ML8.17 AND NOT %ML8.18 AND %ML0.62;
(* /////  QT 이글루 TVL OPEN ///// *)
(* Rung L16 *)
%WW1502 := %WW1600;
(* Rung L19 *)
%ML408.0 := %WW1502 >= 3;
%ML408.1 := %WW1502 > 0;

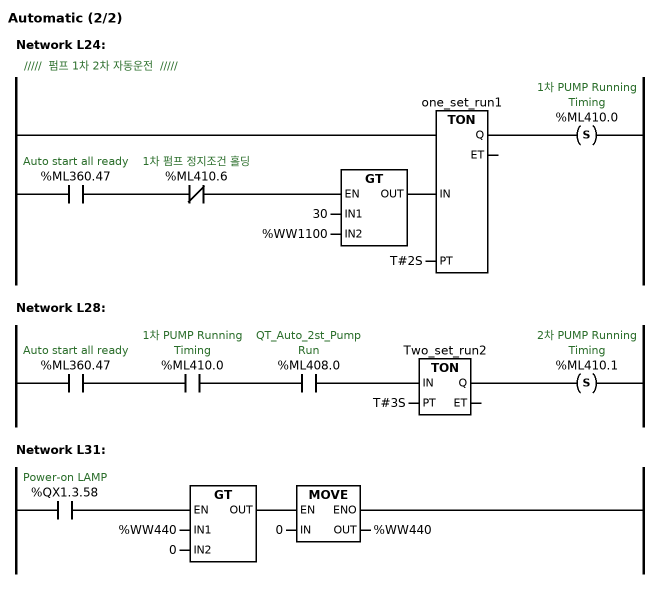
(* /////  펌프 1차 2차 자동운전  ///// *)
(* Rung L24 *)
IF %ML360.47 AND NOT %ML410.6 THEN _t3 := 30 > %WW1100; END_IF;
one_set_run1(IN := _t3, PT := T#2S);
IF one_set_run1.Q THEN %ML410.0 := TRUE; END_IF;
(* Rung L28 *)
Two_set_run2(IN := %ML360.47 AND %ML410.0 AND %ML408.0, PT := T#3S);
IF Two_set_run2.Q THEN %ML410.1 := TRUE; END_IF;
(* Rung L31 *)
IF %QX1.3.58 THEN _t4 := %WW440 > 0; END_IF;
IF _t4 THEN %WW440 := 0; END_IF;

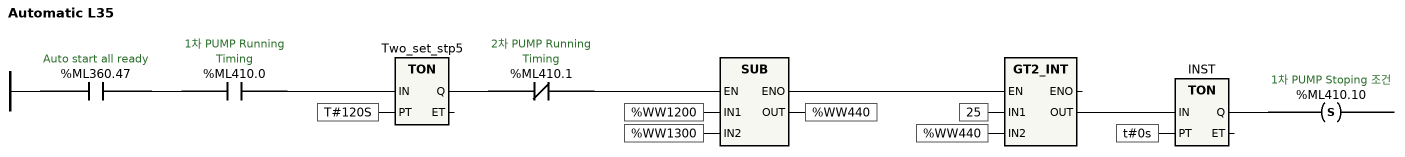
(* Rung L35 *)
Two_set_stp5(IN := %ML360.47 AND %ML410.0, PT := T#120S);
IF Two_set_stp5.Q AND NOT %ML410.1 THEN
    %WW440 := %WW1200 - %WW1300;
    _t5 := GT2_INT(25, %WW440);
END_IF;
INST(IN := _t5, PT := t#0s);
IF INST.Q THEN %ML410.10 := TRUE; END_IF;

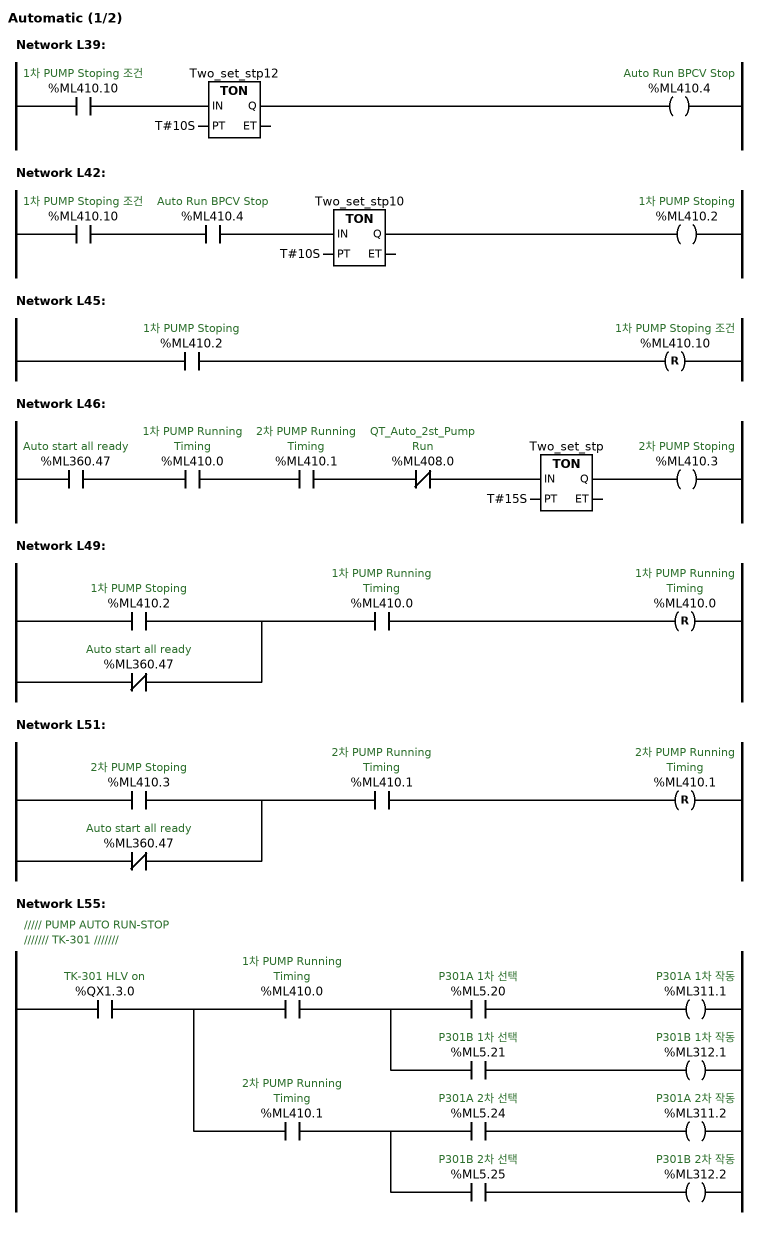
(* Rung L39 *)
Two_set_stp12(IN := %ML410.10, PT := T#10S);
%ML410.4 := Two_set_stp12.Q;
(* Rung L42 *)
Two_set_stp10(IN := %ML410.10 AND %ML410.4, PT := T#10S);
%ML410.2 := Two_set_stp10.Q;
(* Rung L45 *)
IF %ML410.2 THEN %ML410.10 := FALSE; END_IF;
(* Rung L46 *)
Two_set_stp(IN := %ML360.47 AND %ML410.0 AND %ML410.1 AND NOT %ML408.0, PT := T#15S);
%ML410.3 := Two_set_stp.Q;
(* Rung L49 *)
IF (%ML410.2 OR NOT %ML360.47) AND %ML410.0 THEN %ML410.0 := FALSE; END_IF;
(* Rung L51 *)
IF (%ML410.3 OR NOT %ML360.47) AND %ML410.1 THEN %ML410.1 := FALSE; END_IF;
(* ///// PUMP AUTO RUN-STOP *)
(* /////// TK-301 /////// *)
(* Rung L55 *)
%ML311.1 := %QX1.3.0 AND %ML410.0 AND %ML5.20;
%ML312.1 := %QX1.3.0 AND %ML410.0 AND %ML5.21;
%ML311.2 := %QX1.3.0 AND %ML410.1 AND %ML5.24;
%ML312.2 := %QX1.3.0 AND %ML410.1 AND %ML5.25;

